     CASE OP_Arr_OP10P[Output_Page_num] OF	
     300: OLine2:= "O10A_SPARE_Q300_1(Q300.1)                   ";
     301: OLine2:= "O10A_BDY_EMPT_CAM_LGHT2_ON(Q301.1)          ";
     302: OLine2:= "O10B_DRUM_RST(Q302.1)                       ";
     303: OLine2:= "O10B_SPARE_Q303_1(Q303.1)                   ";
     304: OLine2:= "O20_SPARE_Q304_1(Q304.1)                    ";
     305: OLine2:= "O30_CAM_LGHT1_ON(Q305.1)                    ";
     306: OLine2:= "O50_SPARE_Q306_1(Q306.1)                    ";
     307: OLine2:= "O70_DRUM_MTR_FWD(Q307.1)                    ";
     308: OLine2:= "O70_BARLIGHT_OP2(Q308.1)                    ";
     309: OLine2:= "O70_SPARE_Q309_1(Q309.1)                    ";
     1050:OLine2:= "O10A_ORING_LH_PUSHR_CYL_REV_FWD(Q1050.1)    ";
     1051:OLine2:= "O10A_ORING_VERT_CYL_DWN(Q1051.1)            ";
     1052:OLine2:= "O10A_DRUM_FEED_AIRPURGE_ON(Q1052.1)         ";
     1053:OLine2:= "O10A_SPARE_Q1053_1(Q1053.1)                 ";
     1060:OLine2:= "O10B_ORING_LH_PUSHR_CYL_REV_FWD(Q1060.1)    ";
     1061:OLine2:= "O10B_ORING_VERT_CYL_DWN(Q1061.1)            ";
     1062:OLine2:= "O10B_SPARE_Q1062_1(Q1062.1)                 ";
     1063:OLine2:= "O10B_SPARE_Q1063_1(Q1063.1)                 ";
     1150:OLine2:= "O20_LH_OIL_SPIN_ON(Q1150.1)                 ";
     1151:OLine2:= "O40_TOOL_CHO_LOCK(Q1151.1)                  ";
     1152:OLine2:= "O50_SPARE_Q1152_1(Q1152.1)                  ";
     1153:OLine2:= "O80_TOOL_CHO_LOCK(Q1153.1)                     ";
     ELSE 
     OLine2 := " ";
     END_CASE
	 Out_Visibility_2:=TRUE;	
    CASE OP_Arr_OP10P[Output_Page_num] OF
	300:  Out_Lamp2:=O10A_SPARE_Q300_1;
	301:  Out_Lamp2:=O10A_BDY_EMPT_CAM_LGHT2_ON_Q301_1;
	302:  Out_Lamp2:=O10B_DRUM_RST_Q302_1;
	303:  Out_Lamp2:=O10B_SPARE_Q303_1;
	304:  Out_Lamp2:=O20_SPARE_Q304_1;
	305:  Out_Lamp2:=O30_CAM_LGHT1_ON_Q305_1;
	306:  Out_Lamp2:=O50_SPARE_Q306_1;
	307:  Out_Lamp2:=O70_DRUM_MTR_FWD_Q307_1;
	308:  Out_Lamp2:=O70_BARLIGHT_OP2_Q308_1;
	309:  Out_Lamp2:=O70_SPARE_Q309_1;
        1050: Out_Lamp2:=O10A_ORING_LH_PUSHR_CYL_REV_FWD_Q1050_1;
	1051: Out_Lamp2:=O10A_ORING_VERT_CYL_DWN_Q1051_1;
	1052: Out_Lamp2:=O50_RH_REJ_CYL_FWD_Q1152_1;
	1053: Out_Lamp2:=O10A_SPARE_Q1053_1;
	1060: Out_Lamp2:=O10B_ORING_LH_PUSHR_CYL_REV_FWD_Q1060_1;
	1061: Out_Lamp2:=O10B_ORING_VERT_CYL_DWN_Q1061_1;
	1062: Out_Lamp2:=O10B_SPARE_Q1062_1;
	1063: Out_Lamp2:=O10B_SPARE_Q1063_1;
	1150: Out_Lamp2:=O20_LH_OIL_SPIN_ON_Q1150_1;
	1151: Out_Lamp2:=O40_TOOL_CHO_LOCK_Q1151_1;
	1152: Out_Lamp2:=O50_RH_REJ_CYL_FWD_Q1152_1;
	1153: Out_Lamp2:=O80_TOOL_CHO_LOCK_Q1153_1;
   ELSE
       Out_Visibility_2:=FALSE;	
   END_CASE 
   
     CASE OP_Arr_OP10P[Output_Page_num] OF	
     300: OLine3:= "O10A_SPARE_Q300_2(Q300.2)		     ";
     301: OLine3:= "O10A_FIRTREE_ORING_CAM_LGHT1_ON(Q301.2)  ";
     302: OLine3:= "O10B_DRUM_EXT_SPEED(Q302.2)              ";
     303: OLine3:= "O10B_FIRTREE_ORING_CAM_LGHT1_ON(Q303.2)  ";
     304: OLine3:= "O20_SPARE_Q304_2(Q304.2)                 ";
     305: OLine3:= "O30_CAM_LGHT2_ON(Q305.2)                 ";
     306: OLine3:= "O50_DRUM_RUN_IND(Q306.2)                 ";
     307: OLine3:= "O70_DRUM_RST(Q307.2)                     ";
     308: OLine3:= "O70_SPARE_Q308_2(Q308.2)                 ";
     309: OLine3:= "O70_SPARE_Q309_2(Q309.2)                 ";
     1050:OLine3:= "O10A_ORING_RH_GRPR_CLSE_OPN(Q1050.2)     ";
     1051:OLine3:= "O10A_LH_FIRTRE_ORING_REJ_CYL_REV(Q1051.2)";
     1052:OLine3:= "O10A_SPARE_Q1052_2(Q1052.2)              ";
     1053:OLine3:= "O10A_SPARE_Q1053_2(Q1053.2)              ";
     1060:OLine3:= "O10B_ORING_RH_GRPR_CLSE_OPN(Q1060.2)     ";
     1061:OLine3:= "O10B_LH_FIRTRE_ORING_REJ_CYL_REV(Q1061.2)";
     1062:OLine3:= "O10B_SPARE_Q1062_2(Q1062.2)              ";
     1063:OLine3:= "O10B_SPARE_Q1063_2(Q1063.2)              ";
     1150:OLine3:= "O20_RH_OIL_DISPN_ON(Q1150_2)             ";
     1151:OLine3:= "O50_LH_GRIP_OPN_CLSE(Q1151.2)            ";
     1152:OLine3:= "O60_TOOL_CHO_UNLOCK(Q1152.2)             ";
     1153:OLine3:= "O30_AIR_PURGE_ON(Q1153.2)                ";
     ELSE
     	OLine3 := " ";
     END_CASE
	 Out_Visibility_3:=TRUE;	
     CASE OP_Arr_OP10P[Output_Page_num] OF
	300:  Out_Lamp3:=O10A_SPARE_Q300_2;
	301:  Out_Lamp3:=O10A_FIRTREE_ORING_CAM_LGHT1_ON_Q301_2;
	302:  Out_Lamp3:=O10B_DRUM_EXT_SPEED_Q302_2;
	303:  Out_Lamp3:=O10B_FIRTREE_ORING_CAM_LGHT1_ON_Q303_2;
	304:  Out_Lamp3:=O20_SPARE_Q304_2;
	305:  Out_Lamp3:=O30_CAM_LGHT2_ON_Q305_2;
	306:  Out_Lamp3:=O50_DRUM_RUN_IND_Q306_2;
	307:  Out_Lamp3:=O70_DRUM_RST_Q307_2;
	308:  Out_Lamp3:=O70_SPARE_Q308_2;
	309:  Out_Lamp3:=O70_SPARE_Q309_2;
    1050: Out_Lamp3:= O10A_ORING_RH_GRPR_CLSE_OPN_Q1050_2;
	1051: Out_Lamp3:=O10A_LH_FIRTRE_ORING_REJ_CYL_REV_Q1051_2;
	1052: Out_Lamp3:=O10A_SPARE_Q1052_2;
	1053: Out_Lamp3:=O10A_SPARE_Q1053_2;
	1060: Out_Lamp3:=O10B_ORING_RH_GRPR_CLSE_OPN_Q1060_2;
	1061: Out_Lamp3:=O10B_LH_FIRTRE_ORING_REJ_CYL_REV_Q1061_2;
	1062: Out_Lamp3:=O10B_SPARE_Q1062_2;
	1063: Out_Lamp3:=O10B_SPARE_Q1063_2;
	1150: Out_Lamp3:=O20_RH_OIL_DISPN_ON_Q1150_2;
	1151: Out_Lamp3:=O50_LH_GRIP_OPN_Q1151_2;
	1152: Out_Lamp3:=O60_TOOL_CHO_UNLOCK_Q1152_2;
	1153: Out_Lamp3:=O30_AIR_PURGE_ON_Q1153_2;
   ELSE
       Out_Visibility_3:=FALSE;	
   END_CASE 
   
     CASE OP_Arr_OP10P[Output_Page_num] OF	
     300: OLine4:= "O10A_SPARE_Q300_3(Q300.3)	           "; 
     301: OLine4:= "O10A_FIRTREE_ORING_CAM_LGHT2_ON(Q301.3)";
     302: OLine4:= "O10A_SPARE_Q302_3(Q302.3)              ";
     303: OLine4:= "O10B_FIRTREE_ORING_CAM_LGHT2_ON(Q303.3)";
     304: OLine4:= "O20_SPARE_Q304_3(Q304.3)               ";
     305: OLine4:= "O30_SPARE_Q305_3(Q305.3)               ";
     306: OLine4:= "O50_CAM_LGHT1_ON(Q306.3)               ";
     307: OLine4:= "O70_DRUM_EXT_SPEED(Q307.3)             ";
     308: OLine4:= "O70_SPARE_Q308_3(Q308.3)               ";
     309: OLine4:= "O70_SPARE_Q309_3(Q309.3)               ";
     1050:OLine4:= "O10A_ORING_RH_PUSHR_CYL_REV_FWD(Q1050.3)";
     1051:OLine4:= "O10A_LH_FIRTRE_ORING_REJ_CYL_FWD(Q1051.3)";
     1052:OLine4:= "O10A_SPARE_Q1052_3(Q1052.3)            ";
     1053:OLine4:= "O10A_SPARE_Q1053_3(Q1053.3)            ";
     1060:OLine4:= "O10B_ORING_RH_PUSHR_CYL_REV_FWD(Q1060.3)";
     1061:OLine4:= "O10B_LH_FIRTRE_ORING_REJ_CYL_FWD(Q1061.3)";
     1062:OLine4:= "O10B_SPARE_Q1062_3(Q1062.3)            ";
     1063:OLine4:= "O10B_SPARE_Q1063_3(Q1063.3)            ";
     1150:OLine4:= "O20_RH_OIL_SPIN_ON(Q1150.3)            ";
     1151:OLine4:= "O50_SPARE_Q1151_3(Q1151.3)             ";
     1152:OLine4:= "O60_TOOL_CHO_LOCK(Q1152.3)             ";
     1153:OLine4:= "O70_SPARE_Q1153_3(Q1153.3)             ";
     ELSE
     	OLine4 := " ";
     END_CASE
       Out_Visibility_4:=TRUE;	
     CASE OP_Arr_OP10P[Output_Page_num] OF
     300:  Out_Lamp4:=O10A_SPARE_Q300_3;
     301:  Out_Lamp4:=O10A_FIRTREE_ORING_CAM_LGHT2_ON_Q301_3;
     302:  Out_Lamp4:=O10A_SPARE_Q302_3_Q302_3;
     303:  Out_Lamp4:=O10B_FIRTREE_ORING_CAM_LGHT2_ON_Q303_3;
     304:  Out_Lamp4:=O20_SPARE_Q304_3;
     305:  Out_Lamp4:=O30_SPARE_Q305_3;
     306:  Out_Lamp4:=O50_CAM_LGHT1_ON_Q306_3;
     307:  Out_Lamp4:=O70_DRUM_EXT_SPEED_Q307_3;
     308:  Out_Lamp4:=O70_SPARE_Q308_3;
     309:  Out_Lamp4:=O70_SPARE_Q309_3;
     1050: Out_Lamp4:=O10A_ORING_RH_PUSHR_CYL_REV_FWD_Q1050_3;
     1051: Out_Lamp4:=O10A_LH_FIRTRE_ORING_REJ_CYL_FWD_Q1051_3;
     1052: Out_Lamp4:=O10A_SPARE_Q1052_3;
     1053: Out_Lamp4:=O10A_SPARE_Q1053_3;
     1060: Out_Lamp4:=O10B_ORING_RH_PUSHR_CYL_REV_FWD_Q1060_3;
     1061: Out_Lamp4:=O10B_LH_FIRTRE_ORING_REJ_CYL_FWD_Q1061_3;
     1062: Out_Lamp4:=O10B_SPARE_Q1062_3;
     1063: Out_Lamp4:=O10B_SPARE_Q1063_3;
     1150: Out_Lamp4:=O20_RH_OIL_SPIN_ON_Q1150_3;
     1151: Out_Lamp4:=O50_LH_GRIP_CLSE_Q1151_3;
     1152: Out_Lamp4:=O60_TOOL_CHO_LOCK_Q1152_3;
     1153: Out_Lamp4:=O30_SPARE_Q1153_3;
     ELSE	
       Out_Visibility_4:=FALSE;	
     END_CASE 
	 
     CASE OP_Arr_OP10P[Output_Page_num] OF	
     300: OLine5:= "O10A_SPARE_Q300_4(Q300.4)	       	     ";
     301: OLine5:= "O10A_ORING_CAM_LGHT1_ON(Q301.4)          ";
     302: OLine5:= "O10B_DRUM_RUN_IND(Q302.4)                ";
     303: OLine5:= "O10B_ORING_CAM_LGHT1_ON(Q303.4)          ";
     304: OLine5:= "O30_DRUM_MTR_FWD(Q304.4)                 ";
     305: OLine5:= "O30_SPARE_Q305_4(Q305.4)                 ";
     306: OLine5:= "O50_CAM_LGHT2_ON(Q306.4)                 ";
     307: OLine5:= "O70_SPARE_Q307_4(Q307.4)                 ";
     308: OLine5:= "O70_SPARE_Q308_4(Q308.4)                 ";
     309: OLine5:= "O70_SPARE_Q309_4(Q309.4)                 ";
     1050:OLine5:= "O10A_ORING_ROTRY_CYL_O_DEG(Q1050.4)      ";
     1051:OLine5:= "O10A_RH_FIRTRE_ORING_REJ_CYL_REV(Q1051.4)";
     1052:OLine5:= "O10A_SPARE_Q1052_4(Q1052.4)              ";
     1053:OLine5:= "O10A_SPARE_Q1053_4(Q1053.4)              ";
     1060:OLine5:= "O10B_ORING_ROTRY_CYL_O_DEG(Q1060.4)      ";
     1061:OLine5:= "O10B_RH_FIRTRE_ORING_REJ_CYL_REV(Q1061.4)";
     1062:OLine5:= "O10B_SPARE_Q1062_4(Q1062.4)              ";
     1063:OLine5:= "O10B_SPARE_Q1063_4(Q1063.4)              ";
     1150:OLine5:= "O30_LH_REJ_CYL_REV(Q1150.4)              ";
     1151:OLine5:= "O50_RH_GRIP_OPN_CLSE(Q1151.4)            ";
     1152:OLine5:= "O70_LH_REJ_CYL_FWD_REV(Q1152.4)          ";
     1153:OLine5:= "O50_AIR_PURGE_ON(Q1153.4)                ";
     ELSE
     	OLine5 := " ";
     END_CASE
         Out_Visibility_5:=TRUE;	
	 CASE OP_Arr_OP10P[Output_Page_num] OF
	      300:  Out_Lamp5:=O10A_SPARE_Q300_4;
	      301:  Out_Lamp5:=O10A_ORING_CAM_LGHT1_ON_Q301_4;
	      302:  Out_Lamp5:=O10B_DRUM_RUN_IND_Q302_4;
	      303:  Out_Lamp5:=O10B_ORING_CAM_LGHT1_ON_Q303_4;
	      304:  Out_Lamp5:=O30_DRUM_MTR_FWD_Q304_4;
	      305:  Out_Lamp5:=O30_SPARE_Q305_4;
	      306:  Out_Lamp5:=O50_CAM_LGHT2_ON_Q306_4;
	      307:  Out_Lamp5:=O70_SPARE_Q307_4;
           308:  Out_Lamp5:=O70_SPARE_Q308_4;
           309:  Out_Lamp5:=O70_SPARE_Q309_4;
	      1050: Out_Lamp5:=O10A_ORING_ROTRY_CYL_O_DEG_Q1050_4;
	      1051: Out_Lamp5:=O10A_RH_FIRTRE_ORING_REJ_CYL_REV_Q1051_4;
	      1052: Out_Lamp5:=O10A_SPARE_Q1052_4;
	      1053: Out_Lamp5:=O10A_SPARE_Q1053_4;
	      1060: Out_Lamp5:=O10B_ORING_ROTRY_CYL_O_DEG_Q1060_4;
	      1061: Out_Lamp5:=O10B_RH_FIRTRE_ORING_REJ_CYL_REV_Q1061_4;
	      1062: Out_Lamp5:=O10B_SPARE_Q1062_4;
	      1063: Out_Lamp5:=O10B_SPARE_Q1063_4;
	      1150: Out_Lamp5:=O30_LH_REJ_CYL_REV_Q1150_4;
	      1151: Out_Lamp5:=O50_RH_GRIP_OPN_Q1151_4;
	      1152: Out_Lamp5:=O70_LH_REJ_CYL_REV_Q1152_4;
	      1153: Out_Lamp5:=O50_AIR_PURGE_ON_Q1153_4;
 	      ELSE
    	        Out_Visibility_5:=FALSE;	
  	      END_CASE
	 
     CASE OP_Arr_OP10P[Output_Page_num] OF	
     300: OLine6:= "O10A_SPARE_Q300_5(Q300.5)					";
     301: OLine6:= "O10A_ORING_CAM_LGHT2_ON(Q301.5)          ";
     302: OLine6:= "O10_TWR_LMP_RD(Q302.5)                  ";
     303: OLine6:= "O10B_ORING_CAM_LGHT2_ON(Q303.5)          ";
     304: OLine6:= "O30_DRUM_RST(Q304.5)                      ";
     305: OLine6:= "O50_DRUM_MTR_FWD(Q305.5)                  ";
     306: OLine6:= "O50_SPARE_Q306_5(Q306.5)                  ";
     307: OLine6:= "O70_DRUM_RUN_IND(Q307.5)                  ";
     308: OLine6:= "O70_SPARE_Q308_5(Q308.5)                  ";
     309: OLine6:= "O70_SPARE_Q309_5(Q309.5)                  ";
     1050:OLine6:= "O10A_ORING_ROTRY_CYL_180_DEG(Q1050.5)     ";
     1051:OLine6:= "O10A_RH_FIRTRE_ORING_REJ_CYL_FWD(Q1051.5) ";
     1052:OLine6:= "O10A_SPARE_Q1052_5(Q1052.5)               ";
     1053:OLine6:= "O10A_SPARE_Q1053_5(Q1053.5)               ";
     1060:OLine6:= "O10B_ORING_ROTRY_CYL_180_DEG(Q1060.5)     ";
     1061:OLine6:= "O10B_RH_FIRTRE_ORING_REJ_CYL_FWD(Q1061.5) ";
     1062:OLine6:= "O10B_SPARE_Q1062_5	(Q1062.5)             ";
     1063:OLine6:= "O10B_SPARE_Q1063_5	(Q1063.5)             ";
     1150:OLine6:= "O30_LH_REJ_CYL_FWD	(Q1150.5)             ";
     1151:OLine6:= "O50_SPARE_Q1151_5	(Q1151.5)             ";
     1152:OLine6:= "O70_SPARE_Q1152_5	(Q1152.5)             ";
     1153:OLine6:= "O70_AIR_PURGE_ON	Q1153.5               ";
     ELSE
     	OLine6 := " ";
     END_CASE
	 
     Out_Visibility_6:=TRUE;	
	 CASE OP_Arr_OP10P[Output_Page_num] OF
	300:  Out_Lamp6:=O10A_SPARE_Q300_5;
	301:  Out_Lamp6:=O10A_ORING_CAM_LGHT2_ON_Q301_5;
	302:  Out_Lamp6:=O10_TWR_LMP_RD_Q302_5;
	303:  Out_Lamp6:=O10B_ORING_CAM_LGHT2_ON_Q303_5;
	304:  Out_Lamp6:=O30_DRUM_RST_Q304_5;
	305:  Out_Lamp6:=O50_DRUM_MTR_FWD_Q305_5;
	306:  Out_Lamp6:=O50_SPARE_Q306_5;
	307:  Out_Lamp6:=O70_DRUM_RUN_IND_Q307_5;
	308:  Out_Lamp6:=O70_SPARE_Q308_5;
	309:  Out_Lamp6:=O70_SPARE_Q309_5;
	1050: Out_Lamp6:=O10A_ORING_ROTRY_CYL_180_DEG_Q1050_5;
	1051: Out_Lamp6:=O10A_RH_FIRTRE_ORING_REJ_CYL_FWD_Q1051_5;
	1052: Out_Lamp6:=O10A_SPARE_Q1052_5;
	1053: Out_Lamp6:=O10A_SPARE_Q1053_5;
	1060: Out_Lamp6:=O10B_ORING_ROTRY_CYL_180_DEG_Q1060_5;
	1061: Out_Lamp6:=O10B_RH_FIRTRE_ORING_REJ_CYL_FWD_Q1061_5;
	1062: Out_Lamp6:=O10B_SPARE_Q1062_5;
	1063: Out_Lamp6:=O10B_SPARE_Q1063_5;
	1150: Out_Lamp6:=O30_LH_REJ_CYL_FWD_Q1150_5;
	1151: Out_Lamp6:=O50_RH_GRIP_CLSE_Q1151_5;
	1152: Out_Lamp6:=O70_LH_REJ_CYL_FWD_Q1152_5;
	1153: Out_Lamp6:=O30_SPARE_Q1153_5;
   ELSE           
       Out_Visibility_6:=FALSE;	
   END_CASE
	 
     CASE OP_Arr_OP10P[Output_Page_num] OF	
     300: OLine7:= "O10_BARLIGHT_OP1(Q300.6)                      ";
     301: OLine7:= "O10A_FIRTREE_ORING_CAMBAR_LGHT1_ON(Q301.6)    ";
     302: OLine7:= "O10_TWR_LMP_GN(Q302.6)                        ";
     303: OLine7:= "O10B_FIRTREE_ORING_CAMBAR_LGHT1_ON(Q303.6)    ";
     304: OLine7:= "O30_DRUM_EXT_SPEED(Q304.6)                    ";
     305: OLine7:= "O50_DRUM_RST(Q305.6)                          ";
     306: OLine7:= "O50_SPARE_Q306_6(Q306.6)                      ";
     307: OLine7:= "O70_CAM_LGHT1_ON(Q307.6)                      ";
     308: OLine7:= "O70_SPARE_Q308_6(Q308.6)                      ";
     309: OLine7:= "O70_SPARE_Q309_6(Q309.6)                      ";
     1050:OLine7:= "O10A_ORING_HORZ_CYL_REV(Q1050.6)              ";
     1051:OLine7:= "O10A_BDY_SING_CYL_CLSE(Q1051.6)               ";
     1052:OLine7:= "O10A_SPARE_Q1052_6(Q1052.6)                   ";
     1053:OLine7:= "O10A_SPARE_Q1053_6(Q1053.6)                   ";
     1060:OLine7:= "O10B_ORING_HORZ_CYL_REV(Q1060.6)              ";
     1061:OLine7:= "O10B_BDY_SING_CYL_CLSE(Q1061.6)               ";
     1062:OLine7:= "O10B_SPARE_Q1062_6(Q1062.6)                   ";
     1063:OLine7:= "O10B_SPARE_Q1063_6(Q1063.6)                   ";
     1150:OLine7:= "O30_RH_REJ_CYL_REV(Q1150.6)                   ";
     1151:OLine7:= "O50_LH_REJ_CYL_FWD_REV(Q1151.6)               ";
     1152:OLine7:= "O70_RH_REJ_CYL_FWD_REV(Q1152.6)               ";
     1153:OLine7:= "O80_SPARE_Q1153_6(Q1153.6)                    ";
     ELSE
     	OLine7 := " ";
     END_CASE
     
	 Out_Visibility_7:=TRUE;	
	 CASE OP_Arr_OP10P[Output_Page_num] OF
	300:  Out_Lamp7:=O10_BARLIGHT_OP1_Q300_6;
	301:  Out_Lamp7:=O10A_FIRTREE_ORING_CAMBAR_LGHT1_ON_Q301_6;
	302:  Out_Lamp7:=O10_TWR_LMP_GN_Q302_6;
	303:  Out_Lamp7:=O10B_FIRTREE_ORING_CAMBAR_LGHT1_ON_Q303_6;
	304:  Out_Lamp7:=O30_DRUM_EXT_SPEED_Q304_6;
	305:  Out_Lamp7:=O50_DRUM_RST_Q305_6;
	306:  Out_Lamp7:=O50_SPARE_Q306_6;
	307:  Out_Lamp7:=O70_CAM_LGHT1_ON_Q307_6;
	308:  Out_Lamp7:=O70_SPARE_Q308_6;
	309:  Out_Lamp7:=O70_SPARE_Q309_6;
	1050: Out_Lamp7:=O10A_ORING_HORZ_CYL_REV_Q1050_6;
	1051: Out_Lamp7:=O10A_BDY_SING_CYL_CLSE_Q1051_6;
	1052: Out_Lamp7:=O10A_SPARE_Q1052_6;
	1053: Out_Lamp7:=O10A_SPARE_Q1053_6;
	1060: Out_Lamp7:=O10B_ORING_HORZ_CYL_REV_Q1060_6;
	1061: Out_Lamp7:=O10B_BDY_SING_CYL_CLSE_Q1061_6;
	1062: Out_Lamp7:=O10B_SPARE_Q1062_6;
	1063: Out_Lamp7:=O10B_SPARE_Q1063_6;
	1150: Out_Lamp7:=O30_RH_REJ_CYL_REV_Q1150_6;
	1151: Out_Lamp7:=O50_LH_REJ_CYL_REV_Q1151_6;
	1152: Out_Lamp7:=O70_RH_REJ_CYL_REV_Q1152_6;
	1153: Out_Lamp7:=O70_AIR_PURGE_ON_Q1153_6;
   ELSE
       Out_Visibility_7:=FALSE;	
   END_CASE 
	 
     CASE OP_Arr_OP10P[Output_Page_num] OF	
     300: OLine8:= "O10_BARLIGHT_OP2(Q300.7)	       ";
     301: OLine8:= "O10A_SPARE_Q301_7(Q301.7)          ";
     302: OLine8:= "O10_TWR_LMP_YELW(Q302.7)           ";
     303: OLine8:= "O10B_SPARE_Q303_7(Q303.7)          ";
     304: OLine8:= "O30_SPARE_Q304_7(Q304.7)           ";
     305: OLine8:= "O50_SPARE_Q305_7(Q305.7)           ";
     306: OLine8:= "O50_BARLIGHT_OP1(Q306.7)           ";
     307: OLine8:= "O70_CAM_LGHT2_ON(Q307.7)           ";
     308: OLine8:= "O70_SPARE_Q308_7(Q308.7)           ";
     309: OLine8:= "O70_SPARE_Q309_7(Q309.7)           ";
     1050:OLine8:= "O10A_ORING_HORZ_CYL_FWD(Q1050.7)   ";
     1051:OLine8:= "O10A_BDY_SING_CYL_OPN(Q1051.7)     ";
     1052:OLine8:= "O10A_SPARE_Q1052_7(Q1052.7)        ";
     1053:OLine8:= "O10A_SPARE_Q1053_7(Q1053.7)        ";
     1060:OLine8:= "O10B_ORING_HORZ_CYL_FWD(Q1060.7)   ";
     1061:OLine8:= "O10B_BDY_SING_CYL_OPN(Q1061.7)     ";
     1062:OLine8:= "O10B_SPARE_Q1062_7(Q1062.7)        ";
     1063:OLine8:= "O10B_SPARE_Q1063_7(Q1063.7)        ";
     1150:OLine8:= "O30_RH_REJ_CYL_FWD(Q1150.7)        ";
     1151:OLine8:= "O50_SPARE_Q1151_7(Q1151.7)         ";
     1152:OLine8:= "O70_SPARE_Q1152_7(Q1152.7)         ";
     1153:OLine8:= "O80_SPARE_Q1153_7(Q1153.7)         ";
     ELSE
     	OLine8 := " ";
     END_CASE
	 Out_Visibility_8:=TRUE;	
	 CASE OP_Arr_OP10P[Output_Page_num] OF
	300:  Out_Lamp8:=O10_BARLIGHT_OP2_Q300_7;
	301:  Out_Lamp8:=O10A_SPARE_Q301_7;
	302:  Out_Lamp8:=O10_TWR_LMP_YELW_Q302_7;
	303:  Out_Lamp8:=O10B_SPARE_Q303_7;
	304:  Out_Lamp8:=O30_SPARE_Q304_7_Q304_7;
	305:  Out_Lamp8:=O50_SPARE_Q305_7;
	306:  Out_Lamp8:=O50_BARLIGHT_OP1_Q306_7;
	307:  Out_Lamp8:=O70_CAM_LGHT2_ON_Q307_7;
	308:  Out_Lamp8:=O70_SPARE_Q308_7;
	309:  Out_Lamp8:=O70_SPARE_Q309_7;
	1050: Out_Lamp8:=O10A_ORING_HORZ_CYL_FWD_Q1050_7;
	1051: Out_Lamp8:=O10A_BDY_SING_CYL_OPN_Q1051_7;
	1052: Out_Lamp8:=O10A_SPARE_Q1052_7;
	1053: Out_Lamp8:=O10A_SPARE_Q1053_7;
	1060: Out_Lamp8:=O10B_ORING_HORZ_CYL_FWD_Q1060_7;
	1061: Out_Lamp8:=O10B_BDY_SING_CYL_OPN_Q1061_7;
	1062: Out_Lamp8:=O10B_SPARE_Q1062_7;
	1063: Out_Lamp8:=O10B_SPARE_Q1063_7;
	1150: Out_Lamp8:=O30_RH_REJ_CYL_FWD_Q1150_7;
	1151: Out_Lamp8:=O50_LH_REJ_CYL_FWD_Q1151_7;
	1152: Out_Lamp8:=O70_RH_REJ_CYL_FWD_Q1152_7;
	1153: Out_Lamp8:=O30_SPARE_Q1153_7;
   ELSE
       Out_Visibility_8:=FALSE;	
   END_CASE  
	 
 2: CASE IP_Arr_OP90P[Input_Page_num] OF
   400:  Line1:= " I90_PMR_FB(I400.0)                   ";
   401:  Line1:= " I90_DOOR7_CLOSE_FB(I401.0)           ";
   402:  Line1:= " I90_DOOR15_CLOSE_FB(I402.0)          ";
   403:  Line1:= " I120_ATC_STN_POKE_YOKE_3(I403.0)     ";
   404:  Line1:="I90_LHS_ESTOP1_FB(I404.0)	      "  ;
   405:  Line1:="I90_XTS_48VSMPS1_DC_OK(I405.0)        " ;
   1200: Line1:= " I90_RET_LH_GRIPR_CYL_CLSE(I1200.0)   ";
   1201: Line1:= " I90_LH_MOVR_SUP_HORZ_CYL_REV(I1201.0)";
   1210: Line1:= " I90_LH1_REJ_SLIDE_REV(I1210.0)       ";
   1211: Line1:= " I90_SPARE_I1211_0(I1211.0)           ";
   1220: Line1:= " I120_PUSH_CYL_REV(I1220.0)           ";
   1221: Line1:= " I120_REJ_BIN_PRSNCE(I1221.0)          ";
   ELSE
     Line1:= " ";	
   END_CASE
   Visibility_1:=TRUE;
   
   CASE IP_Arr_OP90P[Input_Page_num] OF
	400: Lamp1:=I90_PMR_FB_I400_0 ;
	401: Lamp1:=I90_DOOR7_CLOSE_FB_I401_0 ;
	402: Lamp1:=I90_DOOR15_CLOSE_FB_I402_0 ;
	403: Lamp1:=I120_ATC_STN_POKE_YOKE_3_I403_0;
	404: Lamp1:=I90_LHS_ESTOP1_FB_I404_0 ;
	405: Lamp1:=I90_XTS_48VSMPS1_DC_OK_I405_0 ;
	1200: Lamp1:=I90_RET_LH_GRIPR_CYL_CLSE_I1200_0 ;
	1201: Lamp1:=I90_LH_MOVR_SUP_HORZ_CYL_REV_I1201_0 ;
	1210: Lamp1:=I90_LH1_REJ_SLIDE_REV_I1210_0;
	1211: Lamp1:=I90_SPARE_I1211_0;
	1220: Lamp1:=I120_PUSH_CYL_REV_I1220_0 ;
	1221: Lamp1:=I120_REJ_BIN_PRSNCE_I1221_0 ;
   ELSE
       Visibility_1:=FALSE;	
   END_CASE
   
   CASE IP_Arr_OP90P[Input_Page_num] OF
   400:  Line2:= " I90_SURGE_ARRES_FB(I400.1)           ";
   401:  Line2:= " I90_DOOR8_CLOSE_FB(I401.1)           ";
   402:  Line2:= " I90_DOOR16_CLOSE_FB(I402.1)          ";
   403:  Line2:= " I120_ATC_STN_POKE_YOKE_4(I403.1)     ";
   404: Line2:="I90_LHS_ESTOP2_FB(I404.1)             " ;
   405: Line2:="I90_XTS_48VSMPS2_DC_OK(I405.1)        " ;
   1200: Line2:= " I90_RET_LH_GRIPR_CYL_OPN(I1200.1)    ";
   1201: Line2:= " I90_LH_MOVR_SUP_HORZ_CYL_FWD(I1201.1)";
   1210: Line2:= " I90_LH1_REJ_SLIDE_FWD(I1210.1)       ";
   1211: Line2:= " I90_SPARE_I1211_1(I1211.1)           ";
   1220: Line2:= " I120_PUSH_CYL_FWD(I1220.1)           ";
   1221: Line2:= " I120_SPARE_I1221_1(I1221.1)          ";
   ELSE
     Line2:= " ";	
   END_CASE
     
   Visibility_2:=TRUE;
   
   CASE IP_Arr_OP90P[Input_Page_num] OF
	400: Lamp2:=I90_SURGE_ARRES_FB_I400_1  ;
	401: Lamp2:=I90_DOOR8_CLOSE_FB_I401_1 ;
	402: Lamp2:=I90_DOOR16_CLOSE_FB_I402_1 ;
	403: Lamp2:=I120_ATC_STN_POKE_YOKE_4_I403_1;
	404: Lamp2:=I90_LHS_ESTOP2_FB_I404_1 ;
	405: Lamp2:=I90_XTS_48VSMPS2_DC_OK_I405_1 ;
	1200:Lamp2:=I90_RET_LH_GRIPR_CYL_OPN_I1200_1;
	1201:Lamp2:=I90_LH_MOVR_SUP_HORZ_CYL_FWD_I1201_1  ;
	1210:Lamp2:=I90_LH1_REJ_SLIDE_FWD_I1210_1;
	1211:Lamp2:=I90_SPARE_I1211_1 ;
	1220:Lamp2:=I120_PUSH_CYL_FWD_I1220_1 ;
	1221:Lamp2:=I120_SPARE_I1221_1 ;
   ELSE
       Visibility_2:=FALSE;	
   END_CASE
   
   CASE IP_Arr_OP90P[Input_Page_num] OF
   400:  Line3:= " I90_DOOR1_CLOSE_FB(I400.2)           ";
   401:  Line3:= " I90_DOOR9_CLOSE_FB(I401.2)           ";
   402:  Line3:= " I110_RESRVR_LW_LVL(I402.2)           ";
   403:  Line3:= " I120_ATC_SLAVE_MODL1(I403.2)         ";
   404:  Line3:= "I90_LHS_ESTOP3_FB(I404.2)             " ;
   405:  Line3:= "I90_XTS_48VSMPS3_DC_OK(I405.2)        " ;
   1200: Line3:= " I90_RET_RH_GRIPR_CYL_CLSE(I1200.2)   ";
   1201: Line3:= " I90_RH_MOVR_SUP_VERT_CYL_DWN(I1201.2)";
   1210: Line3:= " I90_RH1_REJ_SLIDE_REV(I1210.2)       ";
   1211: Line3:= " I90_SPARE_I1211_2(I1211.2)           ";
   1220: Line3:= " I120_LH_SING_CYL_REV(I1220.2)        ";
   1221: Line3:= " I120_SPARE_I1221_2(I1221.2)          ";
   ELSE
     Line3:= " ";	
   END_CASE
  
    Visibility_3:=TRUE;
   
   CASE IP_Arr_OP90P[Input_Page_num] OF
	400: Lamp3:=I90_DOOR1_CLOSE_FB_I400_2  ;
	401: Lamp3:=I90_DOOR9_CLOSE_FB_I401_2 ;
	402: Lamp3:=I110_RESRVR_LW_LVL_I402_2 ;
	403: Lamp3:=I120_ATC_SLAVE_MODL1_I403_2 ;
	404: Lamp3:=I90_LHS_ESTOP3_FB_I404_2 ;
	405: Lamp3:=I90_XTS_48VSMPS3_DC_OK_I405_2;
	1200:Lamp3:=I90_RET_RH_GRIPR_CYL_CLSE_I1200_2;
	1201:Lamp3:=I90_RH_MOVR_SUP_VERT_CYL_DWN_I1201_2 ;
	1210:Lamp3:=I90_RH1_REJ_SLIDE_REV_I1210_2 ;
	1211:Lamp3:=I90_SPARE_I1211_2;
	1220:Lamp3:=I120_LH_SING_CYL_REV_I1220_2 ;
	1221:Lamp3:=I120_SPARE_I1221_2 ;
   ELSE
       Visibility_3:=FALSE;	
   END_CASE
     
   CASE IP_Arr_OP90P[Input_Page_num] OF
   400:  Line4:= " I90_DOOR2_CLOSE_FB(I400.3)          ";
   401:  Line4:= " I90_DOOR10_CLOSE_FB(I401.3)         ";
   402:  Line4:= " I110_OILTANK_PRES_SW_FB(I402.3)     ";
   403:  Line4:= " I120_ATC_SLAVE_MODL2(I403.3)        ";
   404:Line4:="I90_RHS_ESTOP1_FB(I404.3)             " ;
   405:Line4:="I90_XTS_24VSMPS_DC_OK(I405.3)         " ;
   1200: Line4:= " I90_RET_RH_GRIPR_CYL_OPN(I1200.3)   ";
   1201: Line4:= " I90_RH_MOVR_SUP_VERT_CYL_UP(I1201.3)";
   1210: Line4:= " I90_RH1_REJ_SLIDE_FWD(I1210.3)      ";
   1211: Line4:= " I90_SPARE_I1211_3(I1211.3)          ";
   1220: Line4:= " I120_LH_SING_CYL_FWD(I1220.3)       ";
   1221: Line4:= " I120_SPARE_I1221_3(I1221.3)         ";
   ELSE
     Line4:= " ";	
   END_CASE
   Visibility_4:=TRUE;
   
   CASE IP_Arr_OP90P[Input_Page_num] OF
	400: Lamp4:=I90_DOOR2_CLOSE_FB_I400_3   ;
	401: Lamp4:=I90_DOOR10_CLOSE_FB_I401_3;
	402: Lamp4:=I110_OILTANK_PRES_SW_FB_I402_3 ;
	403: Lamp4:=I120_ATC_SLAVE_MODL2_I403_3 ;
	404: Lamp4:=I90_RHS_ESTOP1_FB_I404_3 ;
	405: Lamp4:=I90_XTS_24VSMPS_DC_OK_I405_3;
	1200:Lamp4:=I90_RET_RH_GRIPR_CYL_OPN_I1200_3;
	1201:Lamp4:=I90_RH_MOVR_SUP_VERT_CYL_UP_I1201_3  ;
	1210:Lamp4:=I90_RH1_REJ_SLIDE_FWD_I1210_3;
	1211:Lamp4:=I90_SPARE_I1211_3 ;
	1220:Lamp4:=I120_LH_SING_CYL_FWD_I1220_3;
	1221:Lamp4:=I120_SPARE_I1221_3  ;
   ELSE
       Visibility_4:=FALSE;	
   END_CASE  
   
   
   CASE IP_Arr_OP90P[Input_Page_num] OF
   400:  Line5:= " I90_DOOR3_CLOSE_FB(I400.4)           ";
   401:  Line5:= " I90_DOOR11_CLOSE_FB(I401.4)          ";
   402:  Line5:= " I120_ATC_DECLAMP_FB(I402.4)          ";
   403:  Line5:= " I120_SPARE_I403_4(I403.4)            ";
   404:Line5:="I90_RHS_ESTOP2_FB(I404.4)             " ;
   405:Line5:="I120_LH_LOCKSPRING_GRPR_CLSE(I405.4)  " ;
   1200: Line5:= " I90_POSTN_SLIDE_CYL_REV(I1200.4)     ";
   1201: Line5:= " I90_RH_MOVR_SUP_HORZ_CYL_REV(I1201.4)";
   1210: Line5:= " I90_LH2_REJ_SLIDE_REV(I1210.4)       ";
   1211: Line5:= " I90_SPARE_I1211_4(I1211.4)           ";
   1220: Line5:= " I120_CAMERA_SLIDE_CYL_REV(I1220.4)";
   1221: Line5:= " I120_SPARE_I1221_4(I1221.4)          ";
   ELSE
     Line5:= " ";	
   END_CASE
      
    Visibility_5:=TRUE;
   
   CASE IP_Arr_OP90P[Input_Page_num] OF
	400: Lamp5:=I90_DOOR3_CLOSE_FB_I400_4   ;
	401: Lamp5:=I90_DOOR11_CLOSE_FB_I401_4;
	402: Lamp5:=I120_ATC_DECLAMP_FB_I402_4 ;
	403: Lamp5:=I120_SPARE_I403_4 ;
	404: Lamp5:=I90_RHS_ESTOP2_FB_I404_4 ;
	405: Lamp5:=I120_LH_LOCKSPRING_GRPR_CLSE_I405_4;
	1200:Lamp5:=I90_POSTN_SLIDE_CYL_REV_I1200_4;
	1201:Lamp5:=I90_RH_MOVR_SUP_HORZ_CYL_REV_I1201_4  ;
	1210:Lamp5:=I90_LH2_REJ_SLIDE_REV_I1210_4;
	1211:Lamp5:=I90_SPARE_I1211_4 ;
	1220:Lamp5:=I120_CAMERA_SLIDE_CYL_REV_I1220_4;
	1221:Lamp5:=I120_SPARE_I1221_4 ;
   ELSE
       Visibility_5:=FALSE;	
   END_CASE  
   
   CASE IP_Arr_OP90P[Input_Page_num] OF
   400:  Line6:= " I90_DOOR4_CLOSE_FB(I400.5)            ";
   401:  Line6:= " I90_DOOR12_CLOSE_FB(I401.5)           ";
   402:  Line6:= " I120_ATC_CLAMP_FB(I402.5)             ";
   403:  Line6:= " I120_SPARE_I403_5(I403.5)              ";
   404:Line6:="I90_RHS_ESTOP3_FB(I404.5)             " ;
   405:Line6:="I120_LH_LOCKSPRING_GRPR_OPN(I405.5)   " ;
   1200: Line6:= " I90_POSTN_SLIDE_CYL_FWD(I1200.5)      ";
   1201: Line6:= " I90_RH_MOVR_SUP_HORZ_CYL_FWD(I1201.5) ";
   1210: Line6:= " I90_LH2_REJ_SLIDE_FWD(I1210.5)        ";
   1211: Line6:= " I90_SPARE_I1211_5(I1211.5)            ";
   1220: Line6:= " I120_CAMERA_SLIDECYL_FWD(I1220.5)  ";
   1221: Line6:= " I120_SPARE_I1221_5(I1221.5)           ";
   ELSE
     Line6:= " ";	
   END_CASE
   
     
  Visibility_6:=TRUE;
   
   CASE IP_Arr_OP90P[Input_Page_num] OF
	400: Lamp6:=I90_DOOR4_CLOSE_FB_I400_5 ;
	401: Lamp6:=I90_DOOR12_CLOSE_FB_I401_5;
	402: Lamp6:=I120_ATC_CLAMP_FB_I402_5 ;
	403: Lamp6:=I120_SPARE_I403_5 ;
	404: Lamp6:=I90_RHS_ESTOP3_FB_I404_5 ;
	405: Lamp6:=I120_LH_LOCKSPRING_GRPR_OPN_I405_5;
	1200:Lamp6:=I90_POSTN_SLIDE_CYL_FWD_I1200_5;
	1201:Lamp6:=I90_RH_MOVR_SUP_HORZ_CYL_FWD_I1201_5  ;
	1210:Lamp6:=I90_LH2_REJ_SLIDE_FWD_I1210_5;
	1211:Lamp6:=I90_SPARE_I1211_5 ;
	1220:Lamp6:=I120_CAMERA_SLIDE_CYL_FWD_I1220_5;
	1221:Lamp6:=I120_SPARE_I1221_5  ;
   ELSE
       Visibility_6:=FALSE;	
   END_CASE  
   CASE IP_Arr_OP90P[Input_Page_num] OF
   400:  Line7:= " I90_DOOR5_CLOSE_FB(I400.6)           ";
   401:  Line7:= " I90_DOOR13_CLOSE_FB(I401.6)          ";
   402:  Line7:= " I120_ATC_STN_POKE_YOKE_1(I402.6)     ";
   403:  Line7:= " I120_SPARE_I403_6(I403.6)            ";
   404:Line7:="I90_SPARE_I404_6(I404.6)              " ;
   405:Line7:="I120_RH_LOCKSPRING_GRPR_CLSE(I405.6)  " ;
   1200: Line7:= " I90_LH_MOVR_SUP_VERT_CYL_DWN(I1200.6)";
   1201: Line7:= " I90_SPARE_I1201_6(I1201.6)           ";
   1210: Line7:= " I90_RH2_REJ_SLIDE_REV(I1210.6)       ";
   1211: Line7:= " I90_SPARE_I1211_6(I1211.6)           ";
   1220: Line7:= " I120_SLAVE1_PRSN_PARK_TRAY(I1220.6)";
   1221: Line7:= " I120_SPARE_I1221_6(I1221.6)          ";
   ELSE
     Line7:= " ";	
   END_CASE
   
    Visibility_7:=TRUE;
   
   CASE IP_Arr_OP90P[Input_Page_num] OF
	400: Lamp7:=I90_DOOR5_CLOSE_FB_I400_6 ;
	401: Lamp7:=I90_DOOR13_CLOSE_FB_I401_6;
	402: Lamp7:=I120_ATC_STN_POKE_YOKE_1_I402_6 ;
	403: Lamp7:=I120_SPARE_I403_6 ;
	404: Lamp7:=I90_SPARE_I404_6 ;
	405: Lamp7:=I120_RH_LOCKSPRING_GRPR_CLSE_I405_6;
	1200:Lamp7:=I90_LH_MOVR_SUP_VERT_CYL_DWN_I1200_6;
	1201:Lamp7:=I90_SPARE_I1201_6  ;
	1210:Lamp7:=I90_RH2_REJ_SLIDE_REV_I1210_6;
	1211:Lamp7:=I90_SPARE_I1211_6 ;
	1220:Lamp7:=I120_SLAVE1_PRSN_PARK_TRAY_I1220_6;
	1221:Lamp7:=I120_SPARE_I1221_6  ;
   ELSE
       Visibility_7:=FALSE;	
   END_CASE  
     
   CASE IP_Arr_OP90P[Input_Page_num] OF
   400:  Line8:= " I90_DOOR6_CLOSE_FB(I400.7)          ";
   401:  Line8:= " I90_DOOR14_CLOSE_FB(I401.7)         ";
   402:  Line8:= " I120_ATC_STN_POKE_YOKE_2(I402.7)    ";
   403:  Line8:= " I90_RESET_FB_I403_7I403.7)            ";
   404:Line8:="I90_SPARE_I404_7(I404.7)              " ;
   405:Line8:="I120_RH_LOCKSPRING_GRPR_OPN(I405.7)   " ;
   1200: Line8:= " I90_LH_MOVR_SUP_VERT_CYL_UP(I1200.7)";
   1201: Line8:= " I90_SPARE_I1201_7(I1201.7)          ";
   1210: Line8:= " I90_RH2_REJ_SLIDE_FWD(I1210.7)      ";
   1211: Line8:= " I90_SPARE_I1211_7(I1211.7)          ";
   1220: Line8:= " I120_SLAVE2_PRSN_PARK_TRAY(I1220.7)";
   1221: Line8:= " I120_SPARE_I1221_7(I1221.7)         ";
   ELSE
     Line8:= " ";	
   END_CASE
   
     Visibility_8:=TRUE;
   
   CASE IP_Arr_OP90P[Input_Page_num] OF
	400: Lamp8:=I90_DOOR6_CLOSE_FB_I400_7 ;
	401: Lamp8:=I90_DOOR14_CLOSE_FB_I401_7;
	402: Lamp8:=I120_ATC_STN_POKE_YOKE_2_I402_7 ;
	403: Lamp8:=I90_RESET_FB_I403_7 ;
	404: Lamp8:=I90_SPARE_I404_7 ;
	405: Lamp8:=I120_RH_LOCKSPRING_GRPR_OPN_I405_7;
	1200:Lamp8:=I90_LH_MOVR_SUP_VERT_CYL_UP_I1200_7;
	1201:Lamp8:=I90_SPARE_I1201_7 ;
	1210:Lamp8:=I90_RH2_REJ_SLIDE_FWD_I1210_7;
	1211:Lamp8:=I90_SPARE_I1211_7 ;
	1220:Lamp8:=I120_SLAVE2_PRSN_PARK_TRAY_I1220_7;
	1221:Lamp8:=I120_SPARE_I1221_7   ;
   ELSE
       Visibility_8:=FALSE;	
   END_CASE  
   
    CASE OP_Arr_OP90P[Output_Page_num] OF
    400:  OLine1:= "O90_VISN_LGHT1_ON(Q400.0)            ";
    401:  OLine1:= "O90_SPARE_Q401_0(Q401.0)             ";
    402:  OLine1:= "O110_SPARE_Q402_0(Q402.0)            ";
    403:  OLine1:= "O120_TWR_LMP_RD(Q403.0)              ";
    1240: OLine1:= "O90_RET_LH_GRIPR_CYL_CLSE(Q1240.0)   ";
    1241: OLine1:= "O90_POSTN_SLIDE_CYL_REV(Q1241.0)     ";
    1242: OLine1:= "O90_RH_MOVR_SUP_HORZ_CYL_REV(Q1242.0)";
    1250: OLine1:= "O90_LH1_REJ_SLIDE_REV(Q1250.0)       ";
    1251: OLine1:= "O90_RH2_REJ_SLIDE_REV(Q1251.0)       ";
    1260: OLine1:= "O110_LH_OIL_DISPN_ON(Q1260.0)        ";
    1261: OLine1:= "O120_TOOL_CHO_UNLOCK(Q1261.0)        ";
    1262: OLine1:= "O120_CAMERA_SLIDE_CYL_REV(Q1262.0)   ";
    ELSE
      OLine1:= " ";	
    END_CASE
    Out_Visibility_1:=TRUE;
    CASE OP_Arr_OP90P[Output_Page_num] OF
	400:  Out_Lamp1:=O90_VISN_LGHT1_ON_Q400_0;
	401:  Out_Lamp1:=O90_SPARE_Q401_0;
	402:  Out_Lamp1:=O110_SPARE_Q402_0;
	403:  Out_Lamp1:=O120_TWR_LMP_RD_Q403_0;
    1240:  Out_Lamp1:=O90_RET_LH_GRIPR_CYL_CLSE_Q1240_0;
    1241:  Out_Lamp1:=O90_POSTN_SLIDE_CYL_REV_Q1241_0;
    1242:  Out_Lamp1:=O90_RH_MOVR_SUP_HORZ_CYL_REV_Q1242_0;
    1250:  Out_Lamp1:=O90_LH1_REJ_SLIDE_REV_Q1250_0;
    1251:  Out_Lamp1:=O90_RH2_REJ_SLIDE_REV_Q1251_0;
    1260:  Out_Lamp1:=O110_LH_OIL_DISPN_ON_Q1260_0;
    1261:  Out_Lamp1:=O120_TOOL_CHO_UNLOCK_Q1261_0;
    1262:  Out_Lamp1:=O120_CAMERA_SLIDECYL_REV_Q1262_0;
   ELSE
       Out_Visibility_1:=FALSE;	
   END_CASE
	
    CASE OP_Arr_OP90P[Output_Page_num] OF
    400:  OLine2:= "O90_VISN_LGHT2_ON(Q400.1)            ";
    401:  OLine2:= "O90_SPARE_Q401_1(Q401.1)             ";
    402:  OLine2:= "O110_SPARE_Q402_1(Q402.1)            ";
    403:  OLine2:= "O120_TWR_LMP_GN(Q403.1)              ";
    1240: OLine2:= "O90_RET_LH_GRIPR_CYL_OPN(Q1240.1)    ";
    1241: OLine2:= "O90_POSTN_SLIDE_CYL_FWD(Q1241.1)     ";
    1242: OLine2:= "O90_RH_MOVR_SUP_HORZ_CYL_FWD(Q1242.1)";
    1250: OLine2:= "O90_LH1_REJ_SLIDE_FWD(Q1250.1)       ";
    1251: OLine2:= "O90_RH2_REJ_SLIDE_FWD(Q1251.1)       ";
    1260: OLine2:= "O110_LH_OIL_SPIN_ON(Q1260.1)         ";
    1261: OLine2:= "O120_TOOL_CHO_LOCK(Q1261.1)          ";
    1262: OLine2:= "O120_CAMERA_SLIDE_CYL_FWD(Q1262.1)   ";
    ELSE
      OLine2:= " ";	
    END_CASE  
  Out_Visibility_2:=TRUE;
   
   CASE OP_Arr_OP90P[Output_Page_num] OF
    400:  Out_Lamp2:=O90_VISN_LGHT2_ON_Q400_1;
    401:  Out_Lamp2:=O90_SPARE_Q401_1;
    402:  Out_Lamp2:=O110_SPARE_Q402_1;
    403:  Out_Lamp2:=O120_TWR_LMP_GN_Q403_1;
   1240:  Out_Lamp2:=O90_RET_LH_GRIPR_CYL_OPN_Q1240_1;
   1241:  Out_Lamp2:=O90_POSTN_SLIDE_CYL_FWD_Q1241_1;
   1242:  Out_Lamp2:=O90_RH_MOVR_SUP_HORZ_CYL_FWD_Q1242_1;
   1250:  Out_Lamp2:=O90_LH1_REJ_SLIDE_FWD_Q1250_1;
   1251:  Out_Lamp2:=O90_RH2_REJ_SLIDE_FWD_Q1251_1;
   1260:  Out_Lamp2:=O110_LH_OIL_SPIN_ON_Q1260_1;
   1261:  Out_Lamp2:=O120_TOOL_CHO_LOCK_Q1261_1;
   1262:  Out_Lamp2:=O120_CAMERA_SLIDECYL_FWD_Q1262_1;
   ELSE
       Out_Visibility_2:=FALSE;	
   END_CASE 
    
    CASE OP_Arr_OP90P[Output_Page_num] OF
    400:  OLine3:= "O90_LH_DOOR_OPN(Q400.2)              ";
    401:  OLine3:= "O90_SPARE_Q401_2(Q401.2)             ";
    402:  OLine3:= "O110_SPARE_Q402_2(Q402.2)            ";
    403:  OLine3:= "O120_TWR_LMP_YELW(Q403.2)            ";
    1240: OLine3:= "O90_RET_RH_GRIPR_CYL_CLSE(Q1240.2)   ";
    1241: OLine3:= "O90_LH_MOVR_SUP_VERT_CYL_DWN(Q1241.2)";
    1242: OLine3:= "O90_SPARE_Q1242_2(Q1242.2)           ";
    1250: OLine3:= "O90_RH1_REJ_SLIDE_REV(Q1250.2)       ";
    1251: OLine3:= "O90_RH_REJ_AIR_PURGE(Q1251.2)        ";
    1260: OLine3:= "O120_RH_OIL_DISPN_ON(Q1260.2)        ";
    1261: OLine3:= "O110_PUSH_CYL_REV(Q1261.2)           ";
    1262: OLine3:= "O120_SPARE_Q1262_2(Q1262.2)          ";
    ELSE
      OLine3:= " ";	
    END_CASE
    
      Out_Visibility_3:=TRUE;	
   CASE OP_Arr_OP90P[Output_Page_num] OF
   400:  Out_Lamp3:=O90_LH_DOOR_OPN_Q400_2;
   401:  Out_Lamp3:=O90_SPARE_Q401_2;
   402:  Out_Lamp3:=O110_SPARE_Q402_2;
   403:  Out_Lamp3:=O120_TWR_LMP_YELW_Q403_2;
   1240:  Out_Lamp3:=O90_RET_RH_GRIPR_CYL_CLSE_Q1240_2;
   1241:  Out_Lamp3:=O90_LH_MOVR_SUP_VERT_CYL_DWN_Q1241_2;
   1242:  Out_Lamp3:=O90_SPARE_Q1242_2;
   1250:  Out_Lamp3:=O90_RH1_REJ_SLIDE_REV_Q1250_2;
   1251:  Out_Lamp3:=O90_RH_REJ_AIR_PURGE_Q1251_2;
   1260:  Out_Lamp3:=O110_RH_OIL_DISPN_ON_Q1260_2;
   1261:  Out_Lamp3:=O120_PUSH_CYL_REV_Q1261_2;
   1262:  Out_Lamp3:=O120_SPARE_Q1262_2;
   ELSE
       Out_Visibility_3:=FALSE;
   END_CASE 
   
    CASE OP_Arr_OP90P[Output_Page_num] OF
    400:  OLine4:= "O90_RH_DOOR_OPN(Q400.3)             ";
    401:  OLine4:= "O90_SPARE_Q401_3(Q401.3)            ";
    402:  OLine4:= "O110_SPARE_Q402_3(Q402.3)           ";
    403:  OLine4:= "O120_TWR_LMP_BUZZ(Q403.3)           ";
    1240: OLine4:= "O90_RET_RH_GRIPR_CYL_OPN(Q1240.3)   ";
    1241: OLine4:= "O90_LH_MOVR_SUP_VERT_CYL_UP(Q1241.3)";
    1242: OLine4:= "O90_SPARE_Q1242_3(Q1242.3)          ";
    1250: OLine4:= "O90_RH1_REJ_SLIDE_FWD(Q1250.3)      ";
    1251: OLine4:= "O90_SPARE_Q1251_3(Q1251.3)          ";
    1260: OLine4:= "O110_RH_OIL_SPIN_ON(Q1260.3)        ";
    1261: OLine4:= "O120_PUSH_CYL_FWD(Q1261.3)          ";
    1262: OLine4:= "O120_SPARE_Q1262_3(Q1262.3)         ";
    ELSE
      OLine4:= " ";	
    END_CASE

    Out_Visibility_4:=TRUE;
   
   CASE OP_Arr_OP90P[Output_Page_num] OF
   400:  Out_Lamp4:=O90_RH_DOOR_OPN_Q400_3;
   401:  Out_Lamp4:=O90_SPARE_Q401_3;
   402:  Out_Lamp4:=O110_SPARE_Q402_3;
   403:  Out_Lamp4:=O120_TWR_LMP_BUZZ_Q403_3;
   1240: Out_Lamp4:=O90_RET_RH_GRIPR_CYL_OPN_Q1240_3;
   1241: Out_Lamp4:=O90_LH_MOVR_SUP_VERT_CYL_UP_Q1241_3;
   1242: Out_Lamp4:=O90_SPARE_Q1242_3;
   1250: Out_Lamp4:=O90_RH1_REJ_SLIDE_FWD_Q1250_3;
   1251: Out_Lamp4:=O90_SPARE_Q1251_3;
   1260: Out_Lamp4:=O110_RH_OIL_SPIN_ON_Q1260_3;
   1261: Out_Lamp4:=O120_PUSH_CYL_FWD_Q1261_3;
   1262: Out_Lamp4:=O120_SPARE_Q1262_3;
   ELSE
       Out_Visibility_4:=FALSE;
   END_CASE 
   
    Out_Visibility_5:=TRUE;
	
    CASE OP_Arr_OP90P[Output_Page_num] OF
    400:  OLine5:= "O90_FRNT_DOOR_OPN(Q400.4)            ";
    401:  OLine5:= "O110_RH_OIL_DISPN_FRL_VLVE_ON(Q401.4) ";
    402:  OLine5:= "O120_VISN_LGHT1_ON(Q402.4)           ";
    403:  OLine5:= "O120_SPARE_Q403_4(Q403.4)            ";
    1240: OLine5:= "O90_POS_LOCK_CYL1_VLVE_1(Q1240.4)    ";
    1241: OLine5:= "O90_LH_MOVR_SUP_HORZ_CYL_REV(Q1241.4)";
    1242: OLine5:= "O90_SPARE_Q1242_4(Q1242.4)           ";
    1250: OLine5:= "O90_SPARE_Q1250_4(Q1250.4)           ";
    1251: OLine5:= "O90_SPARE_Q1251_4(Q1251.4)           ";
    1260: OLine5:= "O120_LH_GRPR_CLSE(Q1260.4)           ";
    1261: OLine5:= "O120_LH_SING_CYL_REV(Q1261.4)        ";
    1262: OLine5:= "O120_SPARE_Q1262_4(Q1262.4)          ";
    ELSE
      OLine5:= " ";	
    END_CASE
	
   CASE OP_Arr_OP90P[Output_Page_num] OF
   400:  Out_Lamp5:=O90_FRNT_DOOR_OPN_Q400_4;
   401:  Out_Lamp5:=O110_RH_OIL_DISPN_FRL_VLVE_ON_Q401_4;
   402:  Out_Lamp5:=O120_VISN_LGHT1_ON_Q402_4;
   403:  Out_Lamp5:=O120_SPARE_Q403_4;
   1240: Out_Lamp5:=O90_POS_LOCK_CYL1_VLVE_1_Q1240_4;
   1241: Out_Lamp5:=O90_LH_MOVR_SUP_HORZ_CYL_REV_Q1241_4;
   1242: Out_Lamp5:=O90_SPARE_Q1242_4;
   1250: Out_Lamp5:=O90_SPARE_Q1250_4;
   1251: Out_Lamp5:=O90_SPARE_Q1251_4;
   1260: Out_Lamp5:=O120_LH_GRPR_CLSE_Q1260_4;
   1261: Out_Lamp5:=O120_LH_SING_CYL_REV_Q1261_4;
   1262: Out_Lamp5:=O120_SPARE_Q1262_4;
   ELSE          
       Out_Visibility_5:=FALSE;
   END_CASE 
   
    Out_Visibility_6:=TRUE;

    
    CASE OP_Arr_OP90P[Output_Page_num] OF
    400:  OLine6:= "O90_BACK_DOOR_OPN(Q400.5)            ";
    401:  OLine6:= "O20_RH_OIL_DISPN_FRL_VLVE_ON(Q401.5)";
    402:  OLine6:= "O120_VISN_LGHT2_ON(Q402.5)           ";
    403:  OLine6:= "O120_SPARE_Q403_5(Q403.5)            ";
    1240: OLine6:= "O90_POS_LOCK_CYL1_VLVE_2(Q1240.5)    ";
    1241: OLine6:= "O90_LH_MOVR_SUP_HORZ_CYL_FWD(Q1241.5)";
    1242: OLine6:= "O90_SPARE_Q1242_5(Q1242.5)           ";
    1250: OLine6:= "O90_LH1_REJ_AIR_PURGE(Q1250.5)       ";
    1251: OLine6:= "O90_SPARE_Q1251_5(Q1251.5)           ";
    1260: OLine6:= "O120_LH_GRPR_OPN(Q1260.5)            ";
    1261: OLine6:= "O120_LH_SING_CYL_FWD(Q1261.5)        ";
    1262: OLine6:= "O120_SPARE_Q1262_5(Q1262.5)          ";
    ELSE
      OLine6:= " ";	
    END_CASE
		
   CASE OP_Arr_OP90P[Output_Page_num] OF
   400:  Out_Lamp6:=O90_BACK_DOOR_OPN_Q400_5;
   401:  Out_Lamp6:=O20_RH_OIL_DISPN_FRL_VLVE_ON_Q401_5;
   402:  Out_Lamp6:=O120_VISN_LGHT2_ON_Q402_5;
   403:  Out_Lamp6:=O120_SPARE_Q403_5;
   1240: Out_Lamp6:=O90_POS_LOCK_CYL1_VLVE_2_Q1240_5;
   1241: Out_Lamp6:=O90_LH_MOVR_SUP_HORZ_CYL_FWD_Q1241_5;
   1242: Out_Lamp6:=O90_SPARE_Q1242_5;
   1250: Out_Lamp6:=O90_LH1_REJ_AIR_PURGE_Q1250_5;
   1251: Out_Lamp6:=O90_SPARE_Q1251_5;
   1260: Out_Lamp6:=O120_LH_GRPR_OPN_Q1260_5;
   1261: Out_Lamp6:=O120_LH_SING_CYL_FWD_Q1261_5;
   1262: Out_Lamp6:= O120_SPARE_Q1262_5;
   ELSE          
       Out_Visibility_6:=FALSE;
   END_CASE 
    
	Out_Visibility_7:=TRUE;
    
    CASE OP_Arr_OP90P[Output_Page_num] OF
    400:  OLine7:= "O90_IPC_P_S(Q400.6)             ";
    401:  OLine7:= "O110_LH_OIL_DISPN_FRL_VLVE_ON(Q401.6) ";
    402:  OLine7:= "O120_BARLIGHT_OP1(Q402.6)            ";
    403:  OLine7:= "O120_SPARE_Q403_6(Q403.6)            ";
    1240: OLine7:= "O90_POS_LOCK_CYL2_VLVE_1(Q1240.6)    ";
    1241: OLine7:= "O90_RH_MOVR_SUP_VERT_CYL_DWN(Q1241.6)";
    1242: OLine7:= "O90_SPARE_Q1242_6(Q1242.6)           ";
    1250: OLine7:= "O90_LH2_REJ_SLIDE_REV(Q1250.6)       ";
    1251: OLine7:= "O90_SPARE_Q1251_6(Q1251.6)           ";
    1260: OLine7:= "O120_LH_REJ_AIR_PURGE(Q1260.6)       ";
    1261: OLine7:= "O120_RH_GRPR_CLSE(Q1261.6)           ";
    1262: OLine7:= "O120_SPARE_Q1262_6(Q1262.6)          ";
    ELSE
      OLine7:= " ";	
    END_CASE
    	
   CASE OP_Arr_OP90P[Output_Page_num] OF
   400:  Out_Lamp7:=O90_IPC_P_S_Q400_6;
   401:  Out_Lamp7:=O110_LH_OIL_DISPN_FRL_VLVE_ON_Q401_6;
   402:  Out_Lamp7:=O120_BARLIGHT_OP1_Q402_6;
   403:  Out_Lamp7:=O120_SPARE_Q403_6;
   1240: Out_Lamp7:=O90_POS_LOCK_CYL2_VLVE_1_Q1240_6;
   1241: Out_Lamp7:=O90_RH_MOVR_SUP_VERT_CYL_DWN_Q1241_6;
   1242: Out_Lamp7:=O90_SPARE_Q1242_6;
   1250: Out_Lamp7:=O90_LH2_REJ_SLIDE_REV_Q1250_6;
   1251: Out_Lamp7:=O90_SPARE_Q1251_6;
   1260: Out_Lamp7:=O120_RH_GRPR_CLSE_Q1260_6;
   1261: Out_Lamp7:=O120_LH_REJ_AIR_PURGE_Q1261_6;
   1262: Out_Lamp7:=O120_SPARE_Q1262_6;
   ELSE
       Out_Visibility_7:=FALSE;
   END_CASE 
   
    CASE OP_Arr_OP90P[Output_Page_num] OF
    400:  OLine8:= "O90_SPARE_Q400_7(Q400.7)            ";
    401:  OLine8:= "O20_LH_OIL_DISPN_FRL_VLVE_ON(Q401.7)";
    402:  OLine8:= "O120_BARLIGHT_OP2(Q402.7)           ";
    403:  OLine8:= "O120_SPARE_Q403_7(Q403.7)           ";
    1240: OLine8:= "O90_POS_LOCK_CYL2_VLVE_2(Q1240.7)   ";
    1241: OLine8:= "O90_RH_MOVR_SUP_VERT_CYL_UP(Q1241.7)";
    1242: OLine8:= "O90_SPARE_Q1242_7(Q1242.7)          ";
    1250: OLine8:= "O90_LH2_REJ_SLIDE_FWD(Q1250.7)      ";
    1251: OLine8:= "O90_SPARE_Q1251_7(Q1251.7)          ";
    1260: OLine8:= "O120_RH_GRPR_OPN(Q1260.7)           ";
    1261: OLine8:= "O120_RH_REJ_AIR_PURGE(Q1261.7)      ";
    1262: OLine8:= "O120_SPARE_Q1262_7(Q1262.7)         ";
    ELSE
      OLine8:= " ";	
    END_CASE
	
    Out_Visibility_8:=TRUE;
   
   CASE OP_Arr_OP90P[Output_Page_num] OF
   400:  Out_Lamp8:=O90_SPARE_Q400_7;
   401:  Out_Lamp8:=O20_LH_OIL_DISPN_FRL_VLVE_ON_Q401_7;
   402:  Out_Lamp8:=O120_BARLIGHT_OP2_Q402_7;
   403:  Out_Lamp8:=O120_SPARE_Q403_7;
   1240: Out_Lamp8:=O90_POS_LOCK_CYL2_VLVE_2_Q1240_7;
   1241: Out_Lamp8:=O90_RH_MOVR_SUP_VERT_CYL_UP_Q1241_7;
   1242: Out_Lamp8:=O90_SPARE_Q1242_7;
   1250: Out_Lamp8:=O90_LH2_REJ_SLIDE_FWD_Q1250_7;
   1251: Out_Lamp8:=O90_SPARE_Q1251_7;
   1260: Out_Lamp8:=O120_RH_GRPR_OPN_Q1260_7;
   1261: Out_Lamp8:=O120_RH_REJ_AIR_PURGE_Q1261_7;
   1262: Out_Lamp8:=O120_SPARE_Q1262_7;
   ELSE           
       Out_Visibility_8:=FALSE;	
   END_CASE   
   
 3: CASE IP_Arr_OP160P[Input_Page_num] OF
    700: Line1:= "I130_LH_ATC_DECLAMP_FB(I700.0)";
    701: Line1:= "I130_RH_ATC_DECLAMP_FB(I701.0)";
    702: Line1:= "I140_ATC1_DECLAMP_FB(I702.0)  ";
    703: Line1:= "I140_SPARE_I703_0(I703.0)     ";
    704: Line1:= "I140_SPARE_I704_0(I704.0)     ";
    705: Line1:= "I140_ATC2_DECLAMP_FB(I705.0)  ";
    706: Line1:= "I140_SPARE_I706_0(I706.0)     ";
    707: Line1:= "I140_SPARE_I707_0(I707.0)     ";
    708: Line1:= "I140_ATC3_DECLAMP_FB(I708.0)  ";
    709: Line1:= "I140_SPARE_I709_0(I709.0)     ";
    710: Line1:= "I140_SPARE_I710_0(I710.0)"     ;
    711: Line1:= "I160_ATC1_STN_POKE_YOKE_1(I711.0)" ;
    712: Line1:= "I160_RH_COMP_PP_GRPR_CLSE(I712.0)" ;
    //713: Line1:="I160_SPARE_I713_0(I713.0)" ;
    714: Line1:= "I10A_DRUM_FEED_ALRM(I714.0)" ;
    715: Line1:= "I160_SPARE_I715_0(I715.0)";
    1300:Line1:= "I130_LH_ROTRY_0_DEG(I1300.0)" ;
    1301:Line1:= "I140_HORZ_SUP1_CYL_REV(I1301.0)" ;
    1310:Line1:= "I140_HORZ_SUP2_CYL_REV(I1310.0)" ;
    1311:Line1:= "I140_VERT_SUP3_CYL_REV(I1311.0)" ;
    1320:Line1:= "I160_SLIDE_CYL_REV(I1320.0)" ;
    1321:Line1:= "I160_SPARE_I1321_0(I1321.0)" ;
    1330:Line1:= "I160_LH_PALLET_LOCK_CYL_UNLOCK(I1330.0)" ;
    1331:Line1:= "I160_REJ_BOX_DOOR_CLSE(I1331.0)";
    ELSE
      Line1:= " ";	
    END_CASE
  Visibility_1:=TRUE;
      
   CASE IP_Arr_OP160P[Input_Page_num] OF
	700: Lamp1:=I130_LH_ATC_DECLAMP_FBI700_0 ;
	701: Lamp1:=I130_RH_ATC_DECLAMP_FBI701_0 ;
	702: Lamp1:=I140_ATC1_DECLAMP_FBI702_0 ;
	703: Lamp1:=I140_SPARE_I703_0 ;
	704: Lamp1:=I140_SPARE_I704_0I704_0  ;
	705: Lamp1:=I140_ATC2_DECLAMP_FBI705_0 ;
	706: Lamp1:=I140_SPARE_I706_0 ;
	707: Lamp1:=I140_SPARE_I707_0 ;
	708: Lamp1:=I140_ATC3_DECLAMP_FBI708_0 ;
	709: Lamp1:=I140_SPARE_I709_0 ;
	710: Lamp1:=I140_SPARE_I710_0 ;
	711: Lamp1:=I160_ATC1_STN_POKE_YOKE_1I711_0 ;
	712: Lamp1:=I160_RH_COMP_PP_GRPR_CLSEI712_0 ;
	//713: Lamp1:=I160_SPARE_I713_0 ;
	714: Lamp1:=I10A_DRUM_FEED_ALRMI714_0 ;
	715: Lamp1:=I160_SPARE_I715_0 ;
	1300:Lamp1:=I130_LH_ROTRY_0_DEGI1300_0 ;
	1301:Lamp1:=I140_HORZ_SUP1_CYL_REVI1301_0 ;
	1310:Lamp1:=I140_HORZ_SUP2_CYL_REVI1310_0 ;
	1311:Lamp1:=I140_VERT_SUP3_CYL_REVI1311_0 ;
	1320:Lamp1:=I160_SLIDE_CYL_REVI1320_0 ;
	1321:Lamp1:=I160_SPARE_I1321_0 ;
	1330:Lamp1:=I160_LH_PALLET_LOCK_CYL_UNLOCKI1330_0 ;
	1331:Lamp1:=I160_REJ_BOX_DOOR_CLSEI1331_0 ;
   ELSE
       Visibility_1:=FALSE;	
   END_CASE
  
    CASE IP_Arr_OP160P[Input_Page_num] OF
    700: Line2:= "I130_LH_ATC_CLAMP_FB(I700.1)";
    701: Line2:= "I130_RH_ATC_CLAMP_FB(I701.1)";
    702: Line2:= "I140_ATC1_CLAMP_FB(I702.1)  ";
    703: Line2:= "I140_SPARE_I703_1(I703.1)   ";
    704: Line2:= "I140_LK_TST_2_PAS(I704.1)   ";
    705: Line2:= "I140_ATC2_CLAMP_FB(I705.1)  ";
    706: Line2:= "I140_LK_TST_3_PAS(I706.1)   ";
    707: Line2:= "I140_LK_TST_4_PAS(I707.1)   ";
    708: Line2:= "I140_ATC3_CLAMP_FB(I708.1)  ";
    709: Line2:= "I140_SPARE_I709_1(I709.1)   ";
    710: Line2:= "I140_LK_TST_6_PAS(I710.1)" ;
    711: Line2:= "I160_ATC1_STN_POKE_YOKE_2(I711.1)" ;
    712: Line2:= "I160_RH_COMP_PP_GRPR_OPN(I712.1)" ;
    //713: Line2:="I160_SPARE_I713_1(I713.1)" ;
    714: Line2:= "I10A_SPARE_I714_1(I714.1)" ;
    715: Line2:= "I160_SPARE_I715_1(I715.1) ";
    1300:Line2:= "I130_LH_ROTRY_180_DEG(I1300.1)" ;
    1301:Line2:= "I140_HORZ_SUP1_CYL_FWD(I1301.1)" ;
    1310:Line2:= "I140_HORZ_SUP2_CYL_FWD(I1310.1)" ;
    1311:Line2:= "I140_VERT_SUP3_CYL_FWD(I1311.1)" ;
    1320:Line2:= "I160_SLIDE_CYL_FWD(I1320.1)" ;
    1321:Line2:= "I160_SPARE_I1321_1(I1321.1)" ;
    1330:Line2:= "I160_LH_PALLET_LOCK_CYL_LOCK(I1330.1)" ;
    1331:Line2:= "I160_SAM_PART_BAG_DOOR_CLSE(I1331.1)" ;
    ELSE
      Line2:= " ";	
    END_CASE
       Visibility_2:=TRUE;

    CASE IP_Arr_OP160P[Input_Page_num] OF
	700: Lamp2:=I130_LH_ATC_CLAMP_FBI700_1 ;
	701: Lamp2:=I130_RH_ATC_CLAMP_FBI701_1 ;
	702: Lamp2:=I140_ATC1_CLAMP_FBI702_1 ;
	703: Lamp2:=I140_SPARE_I703_1 ;
	704: Lamp2:=I140_LK_TST_2_PASI704_1  ;
	705: Lamp2:=I140_ATC2_CLAMP_FBI705_1 ;
	706: Lamp2:=I140_LK_TST_3_PASI706_1 ;
	707: Lamp2:=I140_LK_TST_4_PASI707_1 ;
	708: Lamp2:=I140_ATC3_CLAMP_FBI708_1 ;
	709: Lamp2:=I140_SPARE_I709_1 ;
	710: Lamp2:=I140_LK_TST_6_PASI710_1 ;
	711: Lamp2:=I160_ATC1_STN_POKE_YOKE_2I711_1 ;
	712: Lamp2:=I160_RH_COMP_PP_GRPR_OPNI712_1 ;
	//713: Lamp2:=I160_SPARE_I713_1 ;
	714: Lamp2:=I10A_SPARE_I714_1 ;
	715: Lamp2:=I160_SPARE_I715_1 ;
	1300:Lamp2:=I130_LH_ROTRY_180_DEGI1300_1 ;
	1301:Lamp2:=I140_HORZ_SUP1_CYL_FWDI1301_1 ;
	1310:Lamp2:=I140_HORZ_SUP2_CYL_FWDI1310_1 ;
	1311:Lamp2:=I140_VERT_SUP3_CYL_FWDI1311_1 ;
	1320:Lamp2:=I160_SLIDE_CYL_FWDI1320_1 ;
	1321:Lamp2:=I160_SPARE_I1321_1 ;
	1330:Lamp2:=I160_LH_PALLET_LOCK_CYL_LOCKI1330_1 ;
	1331:Lamp2:=I160_SAM_PART_BAG_DOOR_CLSEI1331_1 ;
   ELSE
       Visibility_2:=FALSE;	
   END_CASE

    CASE IP_Arr_OP160P[Input_Page_num] OF
    700: Line3:= "I130_LH_ATC_STN_POKE_YOKE_1(I700.2)";
    701: Line3:= "I130_RH_ATC_STN_POKE_YOKE_1(I701.2)";
    702: Line3:= "I140_ATC1_STN_POKE_YOKE_1(I702.2)  ";
    703: Line3:= "I140_SPARE_I703_2(I703.2)          ";
    704: Line3:= "I140_LK_TST_2_FL(I704.2)           ";
    705: Line3:= "I140_ATC2_STN_POKE_YOKE_1(I705.2)  ";
    706: Line3:= "I140_LK_TST_3_FL(I706.2)           ";
    707: Line3:= "I140_LK_TST_4_FL(I707.2)           ";
    708: Line3:= "I140_ATC3_STN_POKE_YOKE_1(I708.2)  ";
    709: Line3:= "I140_SPARE_I709_2(I709.2)          ";
    710: Line3:= "I140_LK_TST_6_FL(I710.2)" ;
    711: Line3:= "I160_ATC1_STN_POKE_YOKE_3(I711.2)" ;
    712: Line3:= "I160_AUTOBAG_READY(I712.2)" ;
    713: Line3:= "I160_VFD_RDY(I713.2)" ;
    714: Line3:= "I10A_DRUM_OFF_ON(I714.2)" ;
    715: Line3:= "I160_SPARE_I715_2(I715.2)" ;
    1300:Line3:= "I130_RH_ROTRY_0_DEG(I1300.2)" ;
    1301:Line3:= "I140_VERT_SUP1_CYL_REV(I1301.2)" ;
    1310:Line3:= "I140_VERT_SUP2_CYL_REV(I1310.2)" ;
    1311:Line3:= "I140_WIPE3_CYL_REV(I1311.2)" ;
    1320:Line3:= "I160_SLAVE1_PRSN_PARK_TRAY(I1320.2)" ;
    1321:Line3:= "I160_SPARE_I1321_2(I1321.2)";
    1330:Line3:= "I160_RH_PALLET_LOCK_CYL_UNLOCK(I1330.2)" ;
    1331:Line3:= "I160_TROLLEY_FIXT_PRSN(I1331.2)" ; 
    ELSE
      Line3:= " ";	
    END_CASE
       Visibility_3:=TRUE;

   CASE IP_Arr_OP160P[Input_Page_num] OF
	700: Lamp3:=I130_LH_ATC_STN_POKE_YOKE_1I700_2 ;
	701: Lamp3:=I130_RH_ATC_STN_POKE_YOKE_1I701_2 ;
	702: Lamp3:=I140_ATC1_STN_POKE_YOKE_1I702_2 ;
	703: Lamp3:=I140_SPARE_I703_2 ;
	704: Lamp3:=I140_LK_TST_2_FLI704_2  ;
	705: Lamp3:=I140_ATC2_STN_POKE_YOKE_1I705_2 ;
	706: Lamp3:=I140_LK_TST_3_FLI706_2 ;
	707: Lamp3:=I140_LK_TST_4_FLI707_2 ;
	708: Lamp3:=I140_ATC3_STN_POKE_YOKE_1I708_2 ;
	709: Lamp3:=I140_SPARE_I709_2 ;
	710: Lamp3:=I140_LK_TST_6_FLI710_2 ;
	711: Lamp3:=I160_ATC1_STN_POKE_YOKE_3I711_2 ;
	712: Lamp3:=I160_AUTOBAG_READYI712_2 ;
	713: Lamp3:=I160_VFD_RDYI713_2 ;
	714: Lamp3:=I10A_DRUM_OFF_ON_I714_2 ;
	715: Lamp3:=I160_SPARE_I715_2 ;
	1300:Lamp3:=I130_RH_ROTRY_0_DEGI1300_2 ;
	1301:Lamp3:=I140_VERT_SUP1_CYL_REVI1301_2 ;
	1310:Lamp3:=I140_VERT_SUP2_CYL_REVI1310_2 ;
	1311:Lamp3:=I140_WIPE3_CYL_REVI1311_2 ;
	1320:Lamp3:=I160_SLAVE1_PRSN_PARK_TRAYI1320_2 ;
	1321:Lamp3:=I160_SPARE_I1321_2 ;
	1330:Lamp3:=I160_RH_PALLET_LOCK_CYL_UNLOCKI1330_2 ;
	1331:Lamp3:=I160_TROLLEY_FIXT_PRSNI1331_2 ;
   ELSE
       Visibility_3:=FALSE;	
   END_CASE

    CASE IP_Arr_OP160P[Input_Page_num] OF
    700: Line4:= "I130_LH_ATC_STN_POKE_YOKE_2(I700.3)";
    701: Line4:= "I130_RH_ATC_STN_POKE_YOKE_2(I701.3)";
    702: Line4:= "I140_ATC1_STN_POKE_YOKE_2(I702.3)  ";
    703: Line4:= "I140_LK_TST_1_PAS(I703.3)          ";
    704: Line4:= "I140_LK_TST_2_REF_PRT_FL(I704.3)   ";
    705: Line4:= "I140_ATC2_STN_POKE_YOKE_2(I705.3)  ";
    706: Line4:= "I140_LK_TST_3_REF_PRT_FL(I706.3)   ";
    707: Line4:= "I140_LK_TST_4_REF_PRT_FL(I707.3)   ";
    708: Line4:= "I140_ATC3_STN_POKE_YOKE_2(I708.3)  ";
    709: Line4:= "I140_LK_TST_5_PAS(I709.3)          ";
    710: Line4:= "I140_LK_TST_6_REF_PRT_FL(I710.3)"   ;
    711: Line4:= "I160_ATC1_STN_POKE_YOKE_4(I711.3)"  ;
    //712: Line4:="I160_SPARE_I712_3(I712.3)"         ;
    713: Line4:= "I160_SPARE_I713_3(I713.3)"          ;
    714: Line4:= "I10A_DRUM_CONV_REV(I714.3)"         ;
    715: Line4:= "I160_SPARE_I715_3(I715.3)"          ;
    1300:Line4:= "I130_RH_ROTRY_180_DEG(I1300.3)"     ;
    1301:Line4:= "I140_VERT_SUP1_CYL_FWD(I1301.3)"    ;
    1310:Line4:= "I140_VERT_SUP2_CYL_FWD(I1310.3)"    ;
    1311:Line4:= "I140_WIPE3_CYL_FWD(I1311.3)"        ;
    1320:Line4:= "I160_SLAVE2_PRSN_PARK_TRAY(I1320.3)" ;
    1321:Line4:= "I160_SPARE_I1321_3(I1321.3)"        ;
    1330:Line4:= "I160_RH_PALLET_LOCK_CYL_LOCK(I1330.3)" ;
    1331:Line4:= "I160_SAM_BOX_DOOR_CLSE(I1331.3)"    ;
    ELSE
      Line4:= " ";	
    END_CASE
       Visibility_4:=TRUE;
   
   CASE IP_Arr_OP160P[Input_Page_num] OF
	700: Lamp4:=I130_LH_ATC_STN_POKE_YOKE_2I700_3 ;
	701: Lamp4:=I130_RH_ATC_STN_POKE_YOKE_2I701_3 ;
	702: Lamp4:=I140_ATC1_STN_POKE_YOKE_2I702_3 ;
	703: Lamp4:=I140_LK_TST_1_PASI703_3 ;
	704: Lamp4:=I140_LK_TST_2_REF_PRT_FLI704_3  ;
	705: Lamp4:=I140_ATC2_STN_POKE_YOKE_2I705_3 ;
	706: Lamp4:=I140_LK_TST_3_REF_PRT_FLI706_3 ;
	707: Lamp4:=I140_LK_TST_4_REF_PRT_FLI707_3 ;
	708: Lamp4:=I140_ATC3_STN_POKE_YOKE_2I708_3 ;
	709: Lamp4:=I140_LK_TST_5_PASI709_3 ;
	710: Lamp4:=I140_LK_TST_6_REF_PRT_FLI710_3 ;
	711: Lamp4:=I160_ATC1_STN_POKE_YOKE_4I711_3 ;
	//712: Lamp4:=I160_SPARE_I712_3 ;
	713: Lamp4:=I160_SPARE_I713_3 ;
	714: Lamp4:=I10A_DRUM_CONV_REV_I714_3 ;
	715: Lamp4:=I160_SPARE_I715_3 ;
	1300:Lamp4:=I130_RH_ROTRY_180_DEGI1300_3 ;
	1301:Lamp4:=I140_VERT_SUP1_CYL_FWDI1301_3 ;
	1310:Lamp4:=I140_VERT_SUP2_CYL_FWDI1310_3 ;
	1311:Lamp4:=I140_WIPE3_CYL_FWDI1311_3 ;
	1320:Lamp4:=I160_SLAVE2_PRSN_PARK_TRAYI1320_3 ;
	1321:Lamp4:=I160_SPARE_I1321_3 ;
	1330:Lamp4:=I160_RH_PALLET_LOCK_CYL_LOCKI1330_3 ;
	1331:Lamp4:=I160_SAM_BOX_DOOR_CLSEI1331_3 ;
   ELSE
       Visibility_4:=FALSE;	
   END_CASE
    
    CASE IP_Arr_OP160P[Input_Page_num] OF
    700: Line5:= "I130_LH_ATC_STN_POKE_YOKE_3(I700.4)";
    701: Line5:= "I130_RH_ATC_STN_POKE_YOKE_3(I701.4)";
    702: Line5:= "I140_ATC1_STN_POKE_YOKE_3(I702.4)  ";
    703: Line5:= "I140_LK_TST_1_FL(I703.4)           ";
    704: Line5:= "I140_LK_TST_2_WARNG(I704.4)        ";
    705: Line5:= "I140_ATC2_STN_POKE_YOKE_3(I705.4)  ";
    706: Line5:= "I140_LK_TST_3_WARNG(I706.4)        ";
    707: Line5:= "I140_LK_TST_4_WARNG(I707.4)        ";
    708: Line5:= "I140_ATC3_STN_POKE_YOKE_3(I708.4)  ";
    709: Line5:= "I140_LK_TST_5_FL(I709.4)           ";
    710: Line5:= "I140_LK_TST_6_WARNG(I710.4)" ;
    711: Line5:= "I160_ATC1_SLAVE_TOOL1(I711.4)" ;
    //712: Line5:="I160_SPARE_I712_4(I712.4)" ;
    713: Line5:= "I160_SPARE_I713_4(I713.4)" ;
    714: Line5:= "I10A_DRUM_CONV_FWD(I714.4)" ;
    715: Line5:= "I160_SPARE_I715_4(I715.4)" ;
    //1300:Line5:="I130_SPARE_I1300_4(I1300.4)" ;
    1301:Line5:= "I140_WIPE1_CYL_REV(I1301.4)" ;
    1310:Line5:= "I140_WIPE2_CYL_REV(I1310.4)" ;
    1311:Line5:= "I140_LEAKTEST_PRESS_SW(I1311.4)" ;
    1320:Line5:= "I160_FIXT_COMP1_PRSN(I1320.4)" ;
    1321:Line5:= "I160_SPARE_I1321_4(I1321.4)" ;
    1330:Line5:= "I160_SPARE_I1330_4(I1330.4)" ;
    1331:Line5:= "I160_SPARE_I1331_4(I1331.4)" ;
    ELSE
      Line5:= " ";	
    END_CASE
       Visibility_5:=TRUE;
   
   CASE IP_Arr_OP160P[Input_Page_num] OF
	700: Lamp5:=I130_LH_ATC_STN_POKE_YOKE_3I700_4 ;
	701: Lamp5:=I130_RH_ATC_STN_POKE_YOKE_3I701_4 ;
	702: Lamp5:=I140_ATC1_STN_POKE_YOKE_3I702_4 ;
	703: Lamp5:=I140_LK_TST_1_FLI703_4 ;
	704: Lamp5:=I140_LK_TST_2_WARNGI704_4  ;
	705: Lamp5:=I140_ATC2_STN_POKE_YOKE_3I705_4 ;
	706: Lamp5:=I140_LK_TST_3_WARNGI706_4 ;
	707: Lamp5:=I140_LK_TST_4_WARNGI707_4 ;
	708: Lamp5:=I140_ATC3_STN_POKE_YOKE_3I708_4 ;
	709: Lamp5:=I140_LK_TST_5_FLI709_4 ;
	710: Lamp5:=I140_LK_TST_6_WARNGI710_4 ;
	711: Lamp5:=I160_ATC1_SLAVE_TOOL1I711_4 ;
	//712: Lamp5:=I160_SPARE_I712_4 ;
	713: Lamp5:=I160_SPARE_I713_4 ;
	714: Lamp5:=I10A_DRUM_CONV_FWD_I714_4 ;
	715: Lamp5:=I160_SPARE_I715_4 ;
	//1300:Lamp5:=I130_SPARE_I1300_4 ;
	1301:Lamp5:=I140_WIPE1_CYL_REVI1301_4 ;
	1310:Lamp5:=I140_WIPE2_CYL_REVI1310_4 ;
	1311:Lamp5:=I140_LEAKTEST_PRESS_SWI1311_4 ;
	1320:Lamp5:=I160_FIXT_COMP1_PRSNI1320_4 ;
	1321:Lamp5:=I160_SPARE_I1321_4 ;
	1330:Lamp5:=I160_SPARE_I1330_4 ;
	1331:Lamp5:=I160_SPARE_I1331_4 ;
   ELSE
       Visibility_5:=FALSE;	
   END_CASE
   
    CASE IP_Arr_OP160P[Input_Page_num] OF
    700: Line6:= "I130_LH_ATC_STN_POKE_YOKE_4(I700.5)";
    701: Line6:= "I130_RH_ATC_STN_POKE_YOKE_4(I701.5)";
    702: Line6:= "I140_ATC1_STN_POKE_YOKE_4(I702.5)  ";
    703: Line6:= "I140_LK_TST_1_REF_PRT_FL(I703.5)   ";
    704: Line6:= "I140_LK_TST_2_END_CYC(I704.5)      ";
    705: Line6:= "I140_ATC2_STN_POKE_YOKE_4(I705.5)  ";
    706: Line6:= "I140_LK_TST_3_END_CYC(I706.5)      ";
    707: Line6:= "I140_LK_TST_4_END_CYC(I707.5)      ";
    708: Line6:= "I140_ATC3_STN_POKE_YOKE_4(I708.5)  ";
    709: Line6:= "I140_LK_TST_5_REF_PRT_FL(I709.5)   ";
    710: Line6:= "I140_LK_TST_6_END_CYC(I710.5)" ;
    711: Line6:= "I160_ATC1_SLAVE_TOOL2(I711.5)" ;
    712: Line6:= "I160_AUTOBAG_ERR_STOP(I712.5)" ;
    713: Line6:= "I160_SPARE_I713_5(I713.5)";
    714: Line6:= "I10A_ROB_MAN_AUTO_MODE(I714.5)" ;
    715: Line6:= "I160_SPARE_I715_5(I715.5)" ;
    //1300:Line6:="I130_SPARE_I1300_5(I1300.5)" ;
    1301:Line6:= "I140_WIPE1_CYL_FWD(I1301.5)" ;
    1310:Line6:= "I140_WIPE2_CYL_FWD(I1310.5)" ;
    1311:Line6:= "I140_SPARE_I1311_5(I1311.5)" ;
    1320:Line6:= "I160_FIXT_COMP2_PRSN(I1320.5)" ;
    1321:Line6:= "I160_SPARE_I1321_5(I1321.5)" ;
    1330:Line6:= "I160_CONV_BDY_PRSN1_SEN(I1330.5)" ;
    1331:Line6:= "I160_SPARE_I1331_5(I1321.5)" ;
    ELSE
      Line6:= " ";	
    END_CASE   
       Visibility_6:=TRUE;
   
   CASE IP_Arr_OP160P[Input_Page_num] OF
	700: Lamp6:=I130_LH_ATC_STN_POKE_YOKE_4I700_5 ;
	701: Lamp6:=I130_RH_ATC_STN_POKE_YOKE_4I701_5 ;
	702: Lamp6:=I140_ATC1_STN_POKE_YOKE_4I702_5 ;
	703: Lamp6:=I140_LK_TST_1_REF_PRT_FLI703_5 ;
	704: Lamp6:=I140_LK_TST_2_END_CYCI704_5  ;
	705: Lamp6:=I140_ATC2_STN_POKE_YOKE_4I705_5 ;
	706: Lamp6:=I140_LK_TST_3_END_CYCI706_5 ;
	707: Lamp6:=I140_LK_TST_4_END_CYCI707_5 ;
	708: Lamp6:=I140_ATC3_STN_POKE_YOKE_4I708_5 ;
	709: Lamp6:=I140_LK_TST_5_REF_PRT_FLI709_5 ;
	710: Lamp6:=I140_LK_TST_6_END_CYCI710_5 ;
	711: Lamp6:=I160_ATC1_SLAVE_TOOL2I711_5 ;
	712: Lamp6:=I160_AUTOBAG_ERR_STOPI712_5 ;
	713: Lamp6:=I160_SPARE_I713_5 ;
	714: Lamp6:=I10A_ROB_MAN_AUTO_MODE_I714_5 ;
	715: Lamp6:=I160_SPARE_I715_5 ;
	//1300:Lamp6:=I130_SPARE_I1300_5 ;
	1301:Lamp6:=I140_WIPE1_CYL_FWDI1301_5 ;
	1310:Lamp6:=I140_WIPE2_CYL_FWDI1310_5 ;
	1311:Lamp6:=I140_SPARE_I1311_5 ;
	1320:Lamp6:=I160_FIXT_COMP2_PRSNI1320_5 ;
	1321:Lamp6:=I160_SPARE_I1321_5 ;
	1330:Lamp6:=I160_CONV_BDY_PRSN1_SENI1330_5 ;
	1331:Lamp6:=I160_SPARE_I1331_5 ;
   ELSE
       Visibility_6:=FALSE;	
   END_CASE
   
    CASE IP_Arr_OP160P[Input_Page_num] OF
    700: Line7:= "I130_LH_ATC_SLAVE_MODL1(I700.6)";
    701: Line7:= "I130_RH_ATC_SLAVE_MODL1(I701.6)";
    702: Line7:= "I140_ATC1_SLAVE_MODL1(I702.6)  ";
    703: Line7:= "I140_LK_TST_1_WARNG(I703.6)    ";
    704: Line7:= "I140_SPARE_I704_6(I704.6)      ";
    705: Line7:= "I140_ATC2_SLAVE_MODL1(I705.6)  ";
    706: Line7:= "I140_SPARE_I706_6(I706.6)      ";
    707: Line7:= "I140_SPARE_I707_6(I707.6)      ";
    708: Line7:= "I140_ATC3_SLAVE_MODL1(I708.6)  ";
    709: Line7:= "I140_LK_TST_5_WARNG(I709.6)    ";
    710: Line7:= "I160_ATC_DECLAMP_FB(I710.6)" ;
    711: Line7:= "I160_FIXT_LH_COMP_PP_GRPR_CLSE(I711.6)" ;
    712: Line7:= "I20_RESRVR_LW_LVL(I712.6)" ;
    713: Line7:= "I160_SPARE_I713_6(I713.6)" ;
    714: Line7:= "I160_SPARE_I714_6(I714.6)" ;
    715: Line7:= "I160_SPARE_I715_6(I715.6)" ;
    //1300:Line7:="I130_SPARE_I1300_6(I1300.6)" ;
    1301:Line7:= "I140_SPARE_I1301_6(I1301.6)" ;
    1310:Line7:= "I140_HORZ_SUP3_CYL_REV(I1310_6)" ;
    1311:Line7:= "I160_MOVR_REM_CYL_REV(I1311_6)" ;
    1320:Line7:= "I160_SPARE_I1320_6(I1320.6)" ;
    1321:Line7:= "I160_SPARE_I1321_6(I1321.6)" ;
    1330:Line7:= "I160_CONV_BDY_PRSN2_SEN(I1330_6)" ;
    1331:Line7:= "I160_SPARE_I1331_6(I1331.6)" ;
    ELSE
      Line7:= " ";	
    END_CASE
       Visibility_7:=TRUE;
   
   CASE IP_Arr_OP160P[Input_Page_num] OF
	700: Lamp7:=I130_LH_ATC_SLAVE_MODL1I700_6 ;
	701: Lamp7:=I130_RH_ATC_SLAVE_MODL1I701_6 ;
	702: Lamp7:=I140_ATC1_SLAVE_MODL1I702_6 ;
	703: Lamp7:=I140_LK_TST_1_WARNGI703_6 ;
	704: Lamp7:=I140_SPARE_I704_6  ;
	705: Lamp7:=I140_ATC2_SLAVE_MODL1I705_6 ;
	706: Lamp7:=I140_SPARE_I706_6 ;
	707: Lamp7:=I140_SPARE_I707_6 ;
	708: Lamp7:=I140_ATC3_SLAVE_MODL1I708_6 ;
	709: Lamp7:=I140_LK_TST_5_WARNGI709_6 ;
	710: Lamp7:=I160_ATC_DECLAMP_FBI710_6 ;
	711: Lamp7:=I160_FIXT_LH_COMP_PP_GRPR_CLSEI711_6 ;
	712: Lamp7:=I20_RESRVR_LW_LVLI712_6 ;
	713: Lamp7:=I160_SPARE_I713_6 ;
	714: Lamp7:=I160_SPARE_I714_6 ;
	715: Lamp7:=I160_SPARE_I715_6 ;
	//1300:Lamp7:=I130_SPARE_I1300_6 ;
	1301:Lamp7:=I140_SPARE_I1301_6 ;
	1310:Lamp7:=I140_HORZ_SUP3_CYL_REVI1310_6 ;
	1311:Lamp7:=I160_MOVR_REM_CYL_REVI1311_6 ;
	1320:Lamp7:=I160_SPARE_I1320_6 ;
	1321:Lamp7:=I160_SPARE_I1321_6 ;
	1330:Lamp7:=I160_CONV_BDY_PRSN2_SENI1330_6 ;
	1331:Lamp7:=I160_SPARE_I1331_6 ;
   ELSE
       Visibility_7:=FALSE;	
   END_CASE
    
    CASE IP_Arr_OP160P[Input_Page_num] OF
    700: Line8:= "I130_LH_ATC_SLAVE_MODL2(I700.7)";
    701: Line8:= "I130_RH_ATC_SLAVE_MODL2(I701.7)";
    702: Line8:= "I140_ATC1_SLAVE_MODL2(I702.7)  ";
    703: Line8:= "I140_LK_TST_1_END_CYC(I703.7)  ";
    704: Line8:= "I140_SPARE_I704.7(I704.7)      ";
    705: Line8:= "I140_ATC2_SLAVE_MODL2(I705.7)  ";
    706: Line8:= "I140_SPARE_I706.7(I706.7)      ";
    707: Line8:= "I140_SPARE_I707.7(I707.7)      ";
    708: Line8:= "I140_ATC3_SLAVE_MODL2(I708.7)  ";
    709: Line8:= "I140_LK_TST_5_END_CYC(I709.7)  ";
    710: Line8:= "I160_ATC_CLAMP_FB(I710.7)" ;
    711: Line8:= "I160_FIXT_LH_COMP_PP_GRPR_OPN(I711.7)" ;
    712: Line8:= "I20_OILTANK_PRES_SW_FB(I712.7)" ;
    713: Line8:= "I160_SPARE_I713_7(I713.7)" ;
    714: Line8:= "I160_SPARE_I714_7(I714.7)" ;
    715: Line8:= "I160_SPARE_I715_7(I715.7)" ;
    //1300:Line8:="I130_SPARE_I1300_7(I1300.7)" ;
    1301:Line8:= "I140_SPARE_I1301_7(I1301.7)" ;
    1310:Line8:= "I140_HORZ_SUP3_CYL_FWD(I1310.7)" ;
    1311:Line8:= "I160_MOVR_REM_CYL_FWD(I1311.7)" ;
    1320:Line8:= "I160_SPARE_I1320_7(I1320.7)" ;
    1321:Line8:= "I160_SPARE_I1321_7(I1321.7)" ;
    1330:Line8:= "I160_SPARE_I1330_7(I1330.7)" ;
    1331:Line8:= "I160_SPARE_I1331_7(I1331.7)" ;
    ELSE
      Line8:= " ";	
    END_CASE
       Visibility_8:=TRUE;
   
   CASE IP_Arr_OP160P[Input_Page_num] OF
	700: Lamp8:=I130_LH_ATC_SLAVE_MODL2I700_7 ;
	701: Lamp8:=I130_RH_ATC_SLAVE_MODL2I701_7 ;
	702: Lamp8:=I140_ATC1_SLAVE_MODL2I702_7 ;
	703: Lamp8:=I140_LK_TST_1_END_CYCI703_7 ;
	704: Lamp8:=I140_SPARE_I704_7  ;
	705: Lamp8:=I140_ATC2_SLAVE_MODL2I705_7 ;
	706: Lamp8:=I140_SPARE_I706_7 ;
	707: Lamp8:=I140_SPARE_I707_7 ;
	708: Lamp8:=I140_ATC3_SLAVE_MODL2I708_7 ;
	709: Lamp8:=I140_LK_TST_5_END_CYCI709_7 ;
	710: Lamp8:=I160_ATC_CLAMP_FBI710_7 ;
	711: Lamp8:=I160_FIXT_LH_COMP_PP_GRPR_OPNI711_7 ;
	712: Lamp8:=I20_OILTANK_PRES_SW_FBI712_7 ;
	713: Lamp8:=I160_SPARE_I713_7 ;
	714: Lamp8:=I160_SPARE_I714_7 ;
	715: Lamp8:=I160_SPARE_I715_7 ;
	//1300:Lamp8:=I130_SPARE_I1300_7 ;
	1301:Lamp8:=I140_SPARE_I1301_7 ;
	1310:Lamp8:=I140_HORZ_SUP3_CYL_FWDI1310_7 ;
	1311:Lamp8:=I160_MOVR_REM_CYL_FWDI1311_7 ;
	1320:Lamp8:=I160_SPARE_I1320_7 ;
	1321:Lamp8:=I160_SPARE_I1321_7 ;
	1330:Lamp8:=I160_SPARE_I1330_7 ;
	1331:Lamp8:=I160_SPARE_I1331_7 ;
   ELSE
       Visibility_8:=FALSE;	
   END_CASE
 
    CASE OP_Arr_OP160P[Output_Page_num] OF
    700: OLine1:= "O140_LK_TST1 _RST(Q700.0)  "; 
    701: OLine1:= "O140_LK_TST1 _SEL7(Q701.0) ";
    702: OLine1:= "O140_LK_TST2 _SEL6(Q702.0) ";
    703: OLine1:= "O140_LK_TST3 _SEL5(Q703.0) ";
    704: OLine1:= "O140_LK_TST4 _SEL4(Q704.0) ";
    705: OLine1:= "O140_LK_TST5 _SEL3(Q705.0) ";
    706: OLine1:= "O140_LK_TST6 _SEL2(Q706.0) ";
    707: OLine1:= "O150_BARLIGHT_OP2(Q707.0)  ";
    708: OLine1:= "O160_VFD_FWD(Q708.0)       ";
    709: OLine1:= "O10A_DRUM_RUN_IND(Q709.0)  ";
    1340: OLine1:= "O130_LH_ROTRY_0_DEG(Q1340.0)";
    1341: OLine1:= "O140_HORZ_SUP1_CYL_REV(Q1341.0)";
    1342: OLine1:= "O140_HORZ_SUP2_CYL_REV(Q1342.0)";
    1343: OLine1:= "O140_HORZ_SUP3_CYL_REV(Q1343.0)";
    1350: OLine1:= "O160_VISN_CHECK_AIR_PURGE(Q1350.0)";
    1351: OLine1:= "O160_TOOL_CHO_UNLOCK(Q1351.0)";
    1352: OLine1:= "O160_SPARE_Q1352_0(Q1352.0)";
    1353: OLine1:= "O160_SPARE_Q1353_0(Q1353.0)";
    ELSE
      OLine1:= " ";	
    END_CASE
       Out_Visibility_1:=TRUE;
   
   CASE OP_Arr_OP160P[Output_Page_num] OF
	700:  Out_Lamp1:=O140_LK_TST1_RST_Q700_0;
	701:  Out_Lamp1:=O140_LK_TST1_SEL7_Q701_0;
	702:  Out_Lamp1:=O140_LK_TST2_SEL6_Q702_0;
	703:  Out_Lamp1:=O140_LK_TST3_SEL5_Q703_0;
	704:  Out_Lamp1:=O140_LK_TST4_SEL4_Q704_0;
	705:  Out_Lamp1:=O140_LK_TST5_SEL3_Q705_0;
	706:  Out_Lamp1:=O140_LK_TST6_SEL2_Q706_0;
	707:  Out_Lamp1:=O150_BARLIGHT_OP2_Q707_0;
	708:  Out_Lamp1:=O160_VFD_FWD_Q708_0;
	709:  Out_Lamp1:=O10A_DRUM_RUN_IND_Q709_0;
	1340:  Out_Lamp1:=O130_LH_ROTRY_0_DEG_Q1340_0;
	1341:  Out_Lamp1:=O140_HORZ_SUP1_CYL_REV_Q1341_0;
	1342:  Out_Lamp1:=O140_HORZ_SUP2_CYL_REV_Q1342_0;
	1343:  Out_Lamp1:=O140_HORZ_SUP3_CYL_REV_Q1343_0;
	1350:  Out_Lamp1:=O160_VISN_CHECK_AIR_PURGE_Q1350_0;
	1351:  Out_Lamp1:=O160_TOOL_CHO_UNLOCK_Q1351_0;
	1352:  Out_Lamp1:=O160_SPARE_Q1352_0;
	1353:  Out_Lamp1:=O160_SPARE_Q1353_0;
   ELSE
       Out_Visibility_1:=FALSE;	
   END_CASE
    
    CASE OP_Arr_OP160P[Output_Page_num] OF
    700: OLine2:= "O140_LK_TST1 _STRT(Q700.1)  ";
    701: OLine2:= "O140_LK_TST2 _RST(Q701.1)   ";
    702: OLine2:= "O140_LK_TST2 _SEL7(Q702.1)  ";
    703: OLine2:= "O140_LK_TST3 _SEL6(Q703.1)  ";
    704: OLine2:= "O140_LK_TST4 _SEL5(Q704.1)  ";
    705: OLine2:= "O140_LK_TST5 _SEL4(Q705.1)  ";
    706: OLine2:= "O140_LK_TST6 _SEL3(Q706.1)  ";
    707: OLine2:= "O160_CHECKER_LGHT_ON(Q707.1)";
    708: OLine2:= "O160_VFD_REV(Q708.1)        ";
    709: OLine2:= "O160_SPARE_Q709.1(Q709.1)   ";
   1340: OLine2:= "O130_LH_ROTRY_180_DEG(Q1340.1)";
   1341: OLine2:= "O140_HORZ_SUP1_CYL_FWD(Q1341.1)";
   1342: OLine2:= "O140_HORZ_SUP2_CYL_FWD(Q1342.1)";
   1343: OLine2:= "O140_HORZ_SUP3_CYL_FWD(Q1343.1)";
   1350: OLine2:= "O160_FIXT_PP_GRPR_CLSE_OPN(Q1350.1)";
   1351: OLine2:= "O160_TOOL_CHO_LOCK(Q1351.1)";
   1352: OLine2:= "O160_SPARE_Q1352_1(Q1352.1)";
   1353: OLine2:= "O160_SPARE_Q1353_1(Q1353.1)";
    ELSE
      OLine2:= " ";	
    END_CASE
       Out_Visibility_2:=TRUE;
   
   CASE OP_Arr_OP160P[Output_Page_num] OF
	700:  Out_Lamp2:=O140_LK_TST1_STRT_Q700_1;
	701:  Out_Lamp2:=O140_LK_TST2_RST_Q701_1;
	702:  Out_Lamp2:=O140_LK_TST2_SEL7_Q702_1;
	703:  Out_Lamp2:=O140_LK_TST3_SEL6_Q703_1;
	704:  Out_Lamp2:=O140_LK_TST4_SEL5_Q704_1;
	705:  Out_Lamp2:=O140_LK_TST5_SEL4_Q705_1;
	706:  Out_Lamp2:=O140_LK_TST6_SEL3_Q706_1;
	707:  Out_Lamp2:=O160_CHECKER_LGHT_ON_Q707_1;
	708:  Out_Lamp2:=O160_VFD_REV_Q708_1;
	709:  Out_Lamp2:=O160_SPARE_Q709_1_Q709_1;
        1340:  Out_Lamp2:=O130_LH_ROTRY_180_DEG_Q1340_1;
	1341:  Out_Lamp2:=O140_HORZ_SUP1_CYL_FWD_Q1341_1;
	1342:  Out_Lamp2:=O140_HORZ_SUP2_CYL_FWD_Q1342_1;
	1343:  Out_Lamp2:=O140_HORZ_SUP3_CYL_FWD_Q1343_1;
	1350:  Out_Lamp2:=O160_FIXT_PP_GRPR_CLSE_OPN_Q1350_1;
	1351:  Out_Lamp2:=O160_TOOL_CHO_LOCK_Q1351_1;
	1352:  Out_Lamp2:=O160_SPARE_Q1352_1;
	1353:  Out_Lamp2:=O160_SPARE_Q1353_1;
   ELSE
       Out_Visibility_2:=FALSE;	
   END_CASE 

    CASE OP_Arr_OP160P[Output_Page_num] OF
    700: OLine3:= "O140_LK_TST1 _SEL1(Q700.2)    ";
    701: OLine3:= "O140_LK_TST2 _STRT(Q701.2)    ";
    702: OLine3:= "O140_LK_TST3 _RST(Q702.2)     ";
    703: OLine3:= "O140_LK_TST3 _SEL7(Q703.2)    ";
    704: OLine3:= "O140_LK_TST4 _SEL6(Q704.2)    ";
    705: OLine3:= "O140_LK_TST5 _SEL5(Q705.2)    ";
    706: OLine3:= "O140_LK_TST6 _SEL4(Q706.2)    ";
    707: OLine3:= "O160_FUME_EXTRTR_ON(Q707.2)   ";
    708: OLine3:= "O160_VFD_STOP(Q708.2)         ";
    709: OLine3:= "O10A_ROB_MAN_AUTO_MODE(Q709.2)";
   1340: OLine3:= "O130_RH_ROTRY_0_DEG(Q1340.2)";
   1341: OLine3:= "O140_VERT_SUP1_CYL_REV(Q1341.2)";
   1342: OLine3:= "O140_VERT_SUP2_CYL_REV(Q1342.2)";
   1343: OLine3:= "O140_VERT_SUP3_CYL_REV(Q1343.2)";
   1350: OLine3:= "O160_LH_COMP_PP_GRPR_CLSE_OPN(Q1350.2)";
   1351: OLine3:= "O160_LH_PALLET_LOCK_CYL_UNLOCK(Q1351.2)";
   1352: OLine3:= "OP160_MOVR_REM_CYL_REV(Q1352.2)";
   1353: OLine3:= "O160_SPARE_Q1353_2(Q1353.2)";
    ELSE
      OLine3:= " ";	
    END_CASE
       Out_Visibility_3:=TRUE;
	
   CASE OP_Arr_OP160P[Output_Page_num] OF
	700:  Out_Lamp3:=O140_LK_TST1_SEL1_Q700_2;
	701:  Out_Lamp3:=O140_LK_TST2_STRT_Q701_2;
	702:  Out_Lamp3:=O140_LK_TST3_RST_Q702_2;
	703:  Out_Lamp3:=O140_LK_TST3_SEL7_Q703_2;
	704:  Out_Lamp3:=O140_LK_TST4_SEL6_Q704_2;
	705:  Out_Lamp3:=O140_LK_TST5_SEL5_Q705_2;
	706:  Out_Lamp3:=O140_LK_TST6_SEL4_Q706_2;
	707:  Out_Lamp3:=O160_FUME_EXTRTR_ON_Q707_2;
	708:  Out_Lamp3:=O160_VFD_STOP_Q708_2;
	709:  Out_Lamp3:=O10A_ROB_MAN_AUTO_MODE_Q709_2;
   1340:  Out_Lamp3:=O130_RH_ROTRY_0_DEG_Q1340_2;
	1341:  Out_Lamp3:=O140_VERT_SUP1_CYL_REV_Q1341_2;
	1342:  Out_Lamp3:=O140_VERT_SUP2_CYL_REV_Q1342_2;
	1343:  Out_Lamp3:=O140_VERT_SUP3_CYL_REV_Q1343_2;
	1350:  Out_Lamp3:=O160_LH_COMP_PP_GRPR_CLSE_OPN_Q1350_2;
	1351:  Out_Lamp3:=O160_LH_PALLET_LOCK_CYL_UNLOCK_Q1351_2;
	1352:  Out_Lamp3:=OP160_MOVR_REM_CYL_REV_Q1352_2;
	1353:  Out_Lamp3:=O160_SPARE_Q1353_2;
   ELSE
       Out_Visibility_3:=FALSE;
   END_CASE 
    
    CASE OP_Arr_OP160P[Output_Page_num] OF
    700: OLine4:= "O140_LK_TST1 _SEL2(Q700.3)    ";
    701: OLine4:= "O140_LK_TST2 _SEL1(Q701.3)    ";
    702: OLine4:= "O140_LK_TST3 _STRT(Q702.3)    ";
    703: OLine4:= "O140_LK_TST4 _RST(Q703.3)     ";
    704: OLine4:= "O140_LK_TST4 _SEL7(Q704.3)    ";
    705: OLine4:= "O140_LK_TST5 _SEL6(Q705.3)    ";
    706: OLine4:= "O140_LK_TST6 _SEL5(Q706.3)    ";
    707: OLine4:= "O160_MC_LMP_ON(Q707.3)        ";
    708: OLine4:= "O160_BOT_MC_LMP_ON(Q708.3)    ";
    709: OLine4:= "O10B_ROB_MAN_AUTO_MODE(Q709.3)";
   1340: OLine4:= "O130_RH_ROTRY_180_DEG(Q1340.3)";
   1341: OLine4:= "O140_VERT_SUP1_CYL_FWD(Q1341.3)";
   1342: OLine4:= "O140_VERT_SUP2_CYL_FWD(Q1342.3)";
   1343: OLine4:= "O140_VERT_SUP3_CYL_FWD(Q1343.3)";
   1350: OLine4:= "O160_RH_COMP_PP_GRPR_CLSE_OPN(Q1350.3)";
   1351: OLine4:= "O160_LH_PALLET_LOCK_CYL_LOCK(Q1351.3)";
   1352: OLine4:= "OP160_MOVR_REM_CYL_FWD(Q1352.3)";
   1353: OLine4:= "O160_SPARE_Q1353_3(Q1353.3)";
    ELSE
      OLine4:= " ";	
    END_CASE
        Out_Visibility_4:=TRUE;
   
   CASE OP_Arr_OP160P[Output_Page_num] OF
	700:  Out_Lamp4:=O140_LK_TST1_SEL2_Q700_3;
	701:  Out_Lamp4:=O140_LK_TST2_SEL1_Q701_3;
	702:  Out_Lamp4:=O140_LK_TST3_STRT_Q702_3;
	703:  Out_Lamp4:=O140_LK_TST4_RST_Q703_3;
	704:  Out_Lamp4:=O140_LK_TST4_SEL7_Q704_3;
	705:  Out_Lamp4:=O140_LK_TST5_SEL6_Q705_3;
	706:  Out_Lamp4:=O140_LK_TST6_SEL5_Q706_3;
	707:  Out_Lamp4:=O160_MC_LMP_ON_Q707_3;
	708:  Out_Lamp4:=O160_BOT_MC_LMP_ON_Q708_3;
	709:  Out_Lamp4:=O10B_ROB_MAN_AUTO_MODE_Q709_3;
	1340: Out_Lamp4:=O130_RH_ROTRY_180_DEG_Q1340_3;
	1341: Out_Lamp4:=O140_VERT_SUP1_CYL_FWD_Q1341_3;
	1342: Out_Lamp4:=O140_VERT_SUP2_CYL_FWD_Q1342_3;
	1343: Out_Lamp4:=O140_VERT_SUP3_CYL_FWD_Q1343_3;
	1350: Out_Lamp4:=O160_RH_COMP_PP_GRPR_CLSE_OPN_Q1350_3;
	1351: Out_Lamp4:=O160_LH_PALLET_LOCK_CYL_LOCK_Q1351_3;
	1352: Out_Lamp4:= OP160_MOVR_REM_CYL_FWD_Q1352_3;
	1353: Out_Lamp4:=O160_SPARE_Q1353_3;
   ELSE
       Out_Visibility_4:=FALSE;
   END_CASE 
    
    CASE OP_Arr_OP160P[Output_Page_num] OF
    700: OLine5:= "O140_LK_TST1 _SEL3(Q700.4)     ";
    701: OLine5:= "O140_LK_TST2 _SEL2(Q701.4)     ";
    702: OLine5:= "O140_LK_TST3 _SEL1(Q702.4)     ";
    703: OLine5:= "O140_LK_TST4 _STRT(Q703.4)     ";
    704: OLine5:= "O140_LK_TST5_RST(Q704.4)       ";
    705: OLine5:= "O140_LK_TST5 _SEL7(Q705.4)     ";
    706: OLine5:= "O140_LK_TST6 _SEL6(Q706.4)     ";
    707: OLine5:= "O160_AUTOBAG_CNT_CMPLTD(Q707.4)";
    708: OLine5:= "O10A_DRUM_MTR_FWD(Q708.4)      ";
    709: OLine5:= "O120_ROB_MAN_AUTO_MODE(Q709.4) ";
   1340: OLine5:= "O130_LH_TOOL_CHO_UNLOCK(Q1340.4)";
   1341: OLine5:= "O140_TOOL1_CHO_UNLOCK(Q1341.4)";
   1342: OLine5:= "O140_TOOL2_CHO_UNLOCK(Q1342.4)";
   1343: OLine5:= "O140_TOOL3_CHO_UNLOCK(Q1343.4)";
   1350: OLine5:= "O160_SLIDE_CYL_REV(Q1350.4)";
   1351: OLine5:= "O160_RH_PALLET_LOCK_CYL_UNLOCK(Q1351.4)";
   1352: OLine5:= "O160_SPARE_Q1352_4(Q1352.4)";
   1353: OLine5:= "O160_SPARE_Q1353_4(Q1353.4)";
    ELSE
      OLine5:= " ";	
    END_CASE
       Out_Visibility_5:=TRUE;
	
    CASE OP_Arr_OP160P[Output_Page_num] OF
	700:  Out_Lamp5:=O140_LK_TST1_SEL3_Q700_4;
	701:  Out_Lamp5:=O140_LK_TST2_SEL2_Q701_4;
	702:  Out_Lamp5:=O140_LK_TST3_SEL1_Q702_4;
	703:  Out_Lamp5:=O140_LK_TST4_STRT_Q703_4;
	704:  Out_Lamp5:=O140_LK_TST5_RST_Q704_4;
	705:  Out_Lamp5:=O140_LK_TST5_SEL7_Q705_4;
	706:  Out_Lamp5:=O140_LK_TST6_SEL6_Q706_4;
	707:  Out_Lamp5:=O160_AUTOBAG_CNT_CMPLTD_Q707_4;
	708:  Out_Lamp5:=O10A_DRUM_MTR_FWD_Q708_4;
	709:  Out_Lamp5:=O120_ROB_MAN_AUTO_MODE_Q709_4;
	1340: Out_Lamp5:=O130_LH_TOOL_CHO_UNLOCK_Q1340_4;
	1341: Out_Lamp5:=O140_TOOL1_CHO_UNLOCK_Q1341_4;
	1342: Out_Lamp5:=O140_TOOL2_CHO_UNLOCK_Q1342_4;
	1343: Out_Lamp5:=O140_TOOL3_CHO_UNLOCK_Q1343_4;
	1350: Out_Lamp5:=O160_SLIDE_CYL_REV_Q1350_4;
	1351: Out_Lamp5:=O160_RH_PALLET_LOCK_CYL_UNLOCK_Q1351_4;
	1352: Out_Lamp5:=O160_SPARE_Q1352_4;
	1353: Out_Lamp5:=O160_SPARE_Q1353_4;
   ELSE
       Out_Visibility_5:=FALSE;
   END_CASE 
    
    CASE OP_Arr_OP160P[Output_Page_num] OF
    700: OLine6:= "O140_LK_TST1 _SEL4(Q700.5)        ";
    701: OLine6:= "O140_LK_TST2 _SEL3(Q701.5)        ";
    702: OLine6:= "O140_LK_TST3 _SEL2(Q702.5)        ";
    703: OLine6:= "O140_LK_TST4 _SEL1(Q703.5)        ";
    704: OLine6:= "O140_LK_TST5 _STRT(Q704.5)        ";
    705: OLine6:= "O140_LK_TST6 _RST(Q705.5)         ";
    706: OLine6:= "O140_LK_TST6 _SEL7(Q706.5)        ";
    707: OLine6:= "O160_SAMPLE_PART_DOR_OPN(Q707.5) ";
    708: OLine6:= "O10A_DRUM_RST(Q708.5)             ";
    709: OLine6:= "O160_SPARE_Q709_5(Q709.5)         ";
   1340: OLine6:= "O130_LH_TOOL_CHO_LOCK(Q1340.5)";
   1341: OLine6:= "O140_TOOL1_CHO_LOCK(Q1341.5)";
   1342: OLine6:= "O140_TOOL2_CHO_LOCK(Q1342.5)";
   1343: OLine6:= "O140_TOOL3_CHO_LOCK(Q1343.5)";
   1350: OLine6:= "O160_SLIDE_CYL_FWD(Q1350.5)";
   1351: OLine6:= "O160_RH_PALLET_LOCK_CYL_LOCK(Q1351.5)";
   1352: OLine6:= "O160_SPARE_Q1352_5(Q1352.5)";
   1353: OLine6:= "O160_SPARE_Q1353_5(Q1353.5)";
    ELSE
      OLine6:= " ";	
    END_CASE
       Out_Visibility_6:=TRUE;
	
    CASE OP_Arr_OP160P[Output_Page_num] OF
	700:  Out_Lamp6:=O140_LK_TST1_SEL4_Q700_5;
	701:  Out_Lamp6:=O140_LK_TST2_SEL3_Q701_5;
	702:  Out_Lamp6:=O140_LK_TST3_SEL2_Q702_5;
	703:  Out_Lamp6:=O140_LK_TST4_SEL1_Q703_5;
	704:  Out_Lamp6:=O140_LK_TST5_STRT_Q704_5;
	705:  Out_Lamp6:=O140_LK_TST6_RST_Q705_5;
	706:  Out_Lamp6:=O140_LK_TST6_SEL7_Q706_5;
	707:  Out_Lamp6:=O160_SAMPLE_PART_DOOR_OPN_Q707_5;
	708:  Out_Lamp6:=O10A_DRUM_RST_Q708_5;
	709:  Out_Lamp6:=O160_SPARE_Q709_5;
	1340: Out_Lamp6:=O130_LH_TOOL_CHO_LOCK_Q1340_5;
	1341: Out_Lamp6:=O140_TOOL1_CHO_LOCK_Q1341_5;
	1342: Out_Lamp6:=O140_TOOL2_CHO_LOCK_Q1342_5;
	1343: Out_Lamp6:=O140_TOOL3_CHO_LOCK_Q1343_5;
	1350: Out_Lamp6:=O160_SLIDE_CYL_FWD_Q1350_5;
	1351: Out_Lamp6:=O160_RH_PALLET_LOCK_CYL_LOCK_Q1351_5;
	1352: Out_Lamp6:=O160_SPARE_Q1352_5;
	1353: Out_Lamp6:=O160_SPARE_Q1353_5;
   ELSE           
       Out_Visibility_6:=FALSE;
   END_CASE 
       
    CASE OP_Arr_OP160P[Output_Page_num] OF
    700: OLine7:= "O140_LK_TST1 _SEL5(Q700.6)    ";
    701: OLine7:= "O140_LK_TST2 _SEL4(Q701.6)    ";
    702: OLine7:= "O140_LK_TST3 _SEL3(Q702.6)    ";
    703: OLine7:= "O140_LK_TST4 _SEL2(Q703.6)    ";
    704: OLine7:= "O140_LK_TST5 _SEL1(Q704.6)    ";
    705: OLine7:= "O140_LK_TST6 _STRT(Q705.6)    ";
    706: OLine7:= "O150_VISN_LGHT_ON(Q706.6)     ";
    707: OLine7:= "O160_REJ_BIN_DOR_OPN(Q707.6) ";
    708: OLine7:= "O10A_DRUM_EXT_SPEED(Q708.6)   ";
    709: OLine7:= "O160_SPARE_Q709_6(Q709.6)     ";
   1340: OLine7:= "O130_RH_TOOL_CHO_UNLOCK(Q1340.6)";
   1341: OLine7:= "O140_WIPE1_CYL_REV(Q1341.6)";
   1342: OLine7:= "O140_WIPE2_CYL_REV(Q1342.6)";
   1343: OLine7:= "O140_WIPE3_CYL_REV(Q1343.6)";
   1350: OLine7:= "O160_SPARE_Q1350_6(Q1350.6)";
   1351: OLine7:= "O160_SPARE_Q1351_6(Q1351.6)";
   1352: OLine7:= "O160_SPARE_Q1352_6(Q1352.6)";
   1353: OLine7:= "O160_SPARE_Q1353_6(Q1353.6)";
    ELSE
      OLine7:= " ";	
    END_CASE
       Out_Visibility_7:=TRUE;
	
   CASE OP_Arr_OP160P[Output_Page_num] OF
	700:  Out_Lamp7:=O140_LK_TST1_SEL5_Q700_6;
	701:  Out_Lamp7:=O140_LK_TST2_SEL4_Q701_6;
	702:  Out_Lamp7:=O140_LK_TST3_SEL3_Q702_6;
	703:  Out_Lamp7:=O140_LK_TST4_SEL2_Q703_6;
	704:  Out_Lamp7:=O140_LK_TST5_SEL1_Q704_6;
	705:  Out_Lamp7:=O140_LK_TST6_STRT_Q705_6;
	706:  Out_Lamp7:=O150_VISN_LGHT_ON_Q706_6;
	707:  Out_Lamp7:=O160_REJ_BIN_DOOR_OPN_Q707_6;
	708:  Out_Lamp7:=O10A_DRUM_EXT_SPEED_Q708_6;
	709:  Out_Lamp7:=O160_SPARE_Q709_6;
	1340: Out_Lamp7:=O130_RH_TOOL_CHO_UNLOCK_Q1340_6;
	1341: Out_Lamp7:=O140_WIPE1_CYL_REV_Q1341_6;
	1342: Out_Lamp7:=O140_WIPE2_CYL_REV_Q1342_6;
	1343: Out_Lamp7:=O140_WIPE3_CYL_REV_Q1343_6;
	1350: Out_Lamp7:=O160_SPARE_Q1350_6;
	1351: Out_Lamp7:=O160_SPARE_Q1351_6;
	1352: Out_Lamp7:=O160_SPARE_Q1352_6;
	1353: Out_Lamp7:=O160_SPARE_Q1353_6;
   ELSE
       Out_Visibility_7:=FALSE;
   END_CASE 
    
    CASE OP_Arr_OP160P[Output_Page_num] OF
    700: OLine8:= "O140_LK_TST1_SEL6(Q700.7)";
    701: OLine8:= "O140_LK_TST2_SEL5(Q701.7)";
    702: OLine8:= "O140_LK_TST3_SEL4(Q702.7)";
    703: OLine8:= "O140_LK_TST4_SEL3(Q703.7)";
    704: OLine8:= "O140_LK_TST5_SEL2(Q704.7)";
    705: OLine8:= "O140_LK_TST6_SEL1(Q705.7)";
    706: OLine8:= "O150_BARLIGHT_OP1(Q706.7) ";
    707: OLine8:= "O160_SPARE(Q707.7)        ";
    708: OLine8:= "O160_SPARE_Q708_7(Q708.7) ";
    709: OLine8:= "O160_SPARE_Q709_7(Q709.7) ";
   1340: OLine8:= "O130_RH_TOOL_CHO_LOCK(Q1340.7)";
   1341: OLine8:= "O140_WIPE1_CYL_FWD(Q1341.7)";
   1342: OLine8:= "O140_WIPE2_CYL_FWD(Q1342.7)";
   1343: OLine8:= "O140_WIPE3_CYL_FWD(Q1343.7)";
   1350: OLine8:= "O160_SPARE_Q1350_7(Q1350.7)";
   1351: OLine8:= "O160_SPARE_Q1351_7(Q1351.7)";
   1352: OLine8:= "O160_SPARE_Q1352_7(Q1352.7)";
   1353: OLine8:= "O160_SPARE_Q1353_7(Q1353.7)";
    ELSE
      OLine8:= " ";	
    END_CASE	
       Out_Visibility_8:=TRUE;
   
   CASE OP_Arr_OP160P[Output_Page_num] OF
	700:  Out_Lamp8:=O140_LK_TST1_SEL6_Q700_7;
	701:  Out_Lamp8:=O140_LK_TST2_SEL5_Q701_7;
	702:  Out_Lamp8:=O140_LK_TST3_SEL4_Q702_7;
	703:  Out_Lamp8:=O140_LK_TST4_SEL3_Q703_7;
	704:  Out_Lamp8:=O140_LK_TST5_SEL2_Q704_7;
	705:  Out_Lamp8:=O140_LK_TST6_SEL1_Q705_7;
	706:  Out_Lamp8:=O150_BARLIGHT_OP1_Q706_7;
	707:  Out_Lamp8:=O160_SPARE_Q707_7;
	708:  Out_Lamp8:=O160_SPARE_Q708_7;
	709:  Out_Lamp8:=O160_SPARE_Q709_7;
	1340: Out_Lamp8:=O130_RH_TOOL_CHO_LOCK_Q1340_7;
	1341: Out_Lamp8:=O140_WIPE1_CYL_FWD_Q1341_7;
	1342: Out_Lamp8:=O140_WIPE2_CYL_FWD_Q1342_7;
	1343: Out_Lamp8:=O140_WIPE3_CYL_FWD_Q1343_7;
	1350: Out_Lamp8:=O160_SPARE_Q1350_7;
	1351: Out_Lamp8:=O160_SPARE_Q1351_7;
	1352: Out_Lamp8:=O160_SPARE_Q1352_7;
	1353: Out_Lamp8:=O160_SPARE_Q1353_7;
   ELSE
       Out_Visibility_8:=FALSE;	
   END_CASE 
  
 4: CASE IP_Arr_OP10A[Input_Page_num] OF
      100:Line1:="I10A_HPR_UNIT_ALRM(I100.0)    ";
      101:Line1:="I10A_HPR_DOOR_SELCTN(I101.0)  ";
      102:Line1:="I10A_LNR_TRK1_CHO_MOD1(I102.0)";
      103:Line1:="I10A_SPARE_I103_0(I103.0)     ";
      ELSE
      	Line1:= " ";
      END_CASE
      
      CASE IP_Arr_OP10A[Input_Page_num] OF
      100:Line2:="I10A_SPARE_I100.1(I100.1)      ";
      101:Line2:="I10A_SPARE_I101.1(I101.1)      ";
      102:Line2:="I10A_LNR_TRK1_CHO_MOD2(I102.1) ";
      103:Line2:="I10A_SPARE_I103_1(I103.1)      ";
      ELSE
      	Line2 := " ";
      END_CASE
      
      CASE IP_Arr_OP10A[Input_Page_num] OF
      100:Line3:="I10A_HPR_LOW_LVL_SEN(I100.2)   ";
      101:Line3:="I10A_BDY_BOWL_LOW_LVL(I101.2)  ";
      102:Line3:="I10A_LNR_TRK2_CHO_MOD1(I102.2) ";
      103:Line3:="I10A_SPARE_I103_2(I103.2)      ";
      ELSE
      	Line3 := " ";
      END_CASE
      
      CASE IP_Arr_OP10A[Input_Page_num] OF
      100:Line4:="I10A_HPR_SOL_DOOR_SW_FB(I100.3)";
      101:Line4:="I10A_BDY_BWL_RUN(I101.3)       ";
      102:Line4:="I10A_LNR_TRK2_CHO_MOD2(I102.3) ";
      103:Line4:="I10A_SPARE_I103_3(I103.3)      ";
      ELSE
      	Line4 := " ";
      END_CASE
      
      CASE IP_Arr_OP10A[Input_Page_num] OF
      100:Line5:="I10A_HPR_OFF_ON(I100.4)";
      101:Line5:="I10A_BDY_LNR1_RUN(I101.4)";
      102:Line5:="I10A_SPARE_I102_4(I102.4)";
      103:Line5:="I10A_SPARE_I103_4(I103.4)";
      ELSE
      	Line5:= " ";
      END_CASE
      
      CASE IP_Arr_OP10A[Input_Page_num] OF
      100:Line6:="I10A_BDY_BOWL_OFF_ON(I100.5)  ";
      101:Line6:="I10A_BDY_LNR2_RUN(I101.5)     ";
      102:Line6:="I10A_SPARE_I102_5(I102.5)";
      103:Line6:="I10A_SPARE_I103_5(I103.5)     ";
      ELSE
      	Line6 := " ";
      END_CASE
      
      CASE IP_Arr_OP10A[Input_Page_num] OF
      100:Line7:="I10A_BDY_LNR1_OFF_ON(I100.6)     ";
      101:Line7:="I10A_BDY_LNR_FEED1_OVRFLW(I101.6)";
      102:Line7:="I10A_LH_BDY_CONT_FB(I102.6)      ";
      103:Line7:="I10A_SPARE_I103_6(I103.6)        ";
      ELSE
      	Line7 := " ";
      END_CASE
      
      CASE IP_Arr_OP10A[Input_Page_num] OF
      100:Line8:="I10A_BDY_LNR2_OFF_ON(I100.7)     ";
      101:Line8:="I10A_BDY_LNR_FEED2_OVRFLW(I101.7)";
      102:Line8:="I10A_RH_BDY_CONT_FB(I102.7)      ";
      103:Line8:="I10A_SPARE_I103_7(I103.7)        ";
      ELSE
      	Line8 := " ";
      END_CASE
	 	Visibility_1:=TRUE;
   
   CASE IP_Arr_OP10A[Input_Page_num] OF
	100: Lamp1:=I10A_HPR_UNIT_ALRM_I100_0 ;
	101: Lamp1:=I10A_HPR_DOOR_SELCTN_I101_0 ;
	102: Lamp1:=I10A_LNR_TRK1_CHO_MOD1_I102_0 ;
	103: Lamp1:=I10A_SPARE_I103_0;
   ELSE
       Visibility_1:=FALSE;	
   END_CASE
   
   Visibility_2:=TRUE;
   
   CASE IP_Arr_OP10A[Input_Page_num] OF
	100: Lamp2:=I10A_SPARE_I100_1 ;
	101: Lamp2:=I10A_SPARE_I101_1;
	102: Lamp2:=I10A_LNR_TRK1_CHO_MOD2_I102_1 ;
	103: Lamp2:=I10A_SPARE_I103_1;
   ELSE
       Visibility_2:=FALSE;	
   END_CASE
   
   
    Visibility_3:=TRUE;
   
   CASE IP_Arr_OP10A[Input_Page_num] OF
	100: Lamp3:=I10A_HPR_LOW_LVL_SEN_I100_2 ;
	101: Lamp3:=I10A_BDY_BOWL_LOW_LVL_I101_2 ;
	102: Lamp3:=I10A_LNR_TRK2_CHO_MOD1_I102_2 ;
	103: Lamp3:=I10A_SPARE_I103_2;
   ELSE
       Visibility_3:=FALSE;	
   END_CASE
   
   
    Visibility_4:=TRUE;
   
   CASE IP_Arr_OP10A[Input_Page_num] OF
	100: Lamp4:=I10A_HPR_SOL_DOOR_SW_FB_I100_3 ;
	101: Lamp4:=I10A_BDY_BWL_RUN_I101_3 ;
	102: Lamp4:=I10A_LNR_TRK2_CHO_MOD2_I102_3 ;
	103: Lamp4:=I10A_SPARE_I103_3;
   ELSE
       Visibility_4:=FALSE;	
   END_CASE
   
   
    
    Visibility_5:=TRUE;
   
   CASE IP_Arr_OP10A[Input_Page_num] OF
	100: Lamp5:=I10A_HPR_OFF_ON_I100_4 ;
	101: Lamp5:=I10A_BDY_LNR1_RUN_I101_4 ;
	102: Lamp5:=I10A_SPARE_I102_4 ;
	103: Lamp5:=I10A_SPARE_I103_4;
   ELSE
       Visibility_5:=FALSE;	
   END_CASE
   
    
    Visibility_6:=TRUE;
   
   CASE IP_Arr_OP10A[Input_Page_num] OF
	100: Lamp6:=I10A_BDY_BOWL_OFF_ON_I100_5 ;
	101: Lamp6:=I10A_BDY_LNR2_RUN_I101_5 ;
	102: Lamp6:=I10A_SPARE_I102_5 ;
	103: Lamp6:=I10A_SPARE_I103_5;
   ELSE
       Visibility_6:=FALSE;	
   END_CASE
   
   
      
    Visibility_7:=TRUE;
   
   CASE IP_Arr_OP10A[Input_Page_num] OF
	100: Lamp7:=I10A_BDY_LNR1_OFF_ON_I100_6 ;
	101: Lamp7:=I10A_BDY_LNR_FEED1_OVRFLW_I101_6 ;
	102: Lamp7:=I10A_LH_BDY_CONT_FB_I102_6;
	103: Lamp7:=I10A_SPARE_I103_6;
   ELSE
       Visibility_7:=FALSE;	
   END_CASE


 	Visibility_8:=TRUE;
   
   CASE IP_Arr_OP10A[Input_Page_num] OF
	100: Lamp8:=I10A_BDY_LNR2_OFF_ON_I100_7 ;
	101: Lamp8:=I10A_BDY_LNR_FEED2_OVRFLW_I101_7 ;
	102: Lamp8:=I10A_RH_BDY_CONT_FB_I102_7 ;
	103: Lamp8:=I10A_SPARE_I103_7;
   ELSE
       Visibility_8:=FALSE;	
   END_CASE

	
	 CASE OP_Arr_OP10A[Output_Page_num] OF
     100:OLine1:="O10A_HPR_MTR_FWD(Q100.0)  ";
     101:OLine1:="O10A_BDY_BOWL_ON(Q101.0)  ";
     102:OLine1:="O10A_SPARE_Q102_0(Q102.0) ";
     103:OLine1:="O10A_SPARE_Q103_0(Q103.0) ";
     ELSE
     	OLine1:= " ";
     END_CASE
     
     CASE OP_Arr_OP10A[Output_Page_num] OF
     100:OLine2:="O10A_HPR_RST(Q100.1)         ";
     101:OLine2:="O10A_BDY_LNR_FEED1_ON(Q101.1)";
     102:OLine2:="O10A_SPARE_Q102_1(Q102.1)    ";
     103:OLine2:="O10A_SPARE_Q103_1(Q103.1)    ";
     ELSE
     	OLine2:= " ";
     END_CASE
     
     CASE OP_Arr_OP10A[Output_Page_num] OF
     100:OLine3:="O10A_EXT_SPEED(Q100.2)       ";
     101:OLine3:="O10A_BDY_LNR_FEED2_ON(Q101.2)";
     102:OLine3:="O10A_SPARE_Q102_2(Q102.2)    ";
     103:OLine3:="O10A_SPARE_Q103_2(Q103.2)    ";
     ELSE
     	OLine3:= " ";
     END_CASE
     
     CASE OP_Arr_OP10A[Output_Page_num] OF
     100:OLine4:="O10A_SPARE_Q100.3(Q100.3)      ";
     101:OLine4:="O10A_BDY_LNR1_AIR_PURGE(Q101.3)";
     102:OLine4:="O10A_SPARE_Q102_3(Q102.3)      ";
     103:OLine4:="O10A_SPARE_Q103_3(Q103.3)      ";
     ELSE
     	OLine4:= " ";
     END_CASE
     
     CASE OP_Arr_OP10A[Output_Page_num] OF
     100:OLine5:="O10A_HPR_DOOR_SELCTN_IND(Q100.4)";
   //101:OLine5:="O10A_BDY_LNR2_AIRPURGE(Q101.4)";
     102:OLine5:="O10A_SPARE_Q102_4(Q102.4)";
     103:OLine5:="O10A_SPARE_Q103_4(Q103.4)";
     ELSE
     	OLine5:= " ";
     END_CASE
     
     CASE OP_Arr_OP10A[Output_Page_num] OF
     100:OLine6:="O10A_HPR_TWR_LMP_RED(Q100.5)";
     101:OLine6:="O10A_HPR_DOOR_OPN(Q101.5)   ";
     102:OLine6:="O10A_SPARE_Q102_5(Q102.5)   ";
     103:OLine6:="O10A_SPARE_Q103_5(Q103.5)   ";
     ELSE
     	OLine6:= " ";
     END_CASE
     
     CASE OP_Arr_OP10A[Output_Page_num] OF
     100:OLine7:="O10A_HPR_TWR_LMP_GREEN(Q100.6)";
     101:OLine7:="O10A_SPARE_Q101_6(Q101.6)     ";
     102:OLine7:="O10A_SPARE_Q102_6(Q102.6)     ";
     103:OLine7:="O10A_SPARE_Q103_6(Q103.6)     ";
     ELSE
     	OLine7:= " ";
     END_CASE
     
     CASE OP_Arr_OP10A[Output_Page_num] OF
     100:OLine8:="O10A_SPARE_Q100_7(Q100.7)";
     101:OLine8:="O10A_SPARE_Q101_7(Q101.7)";
     102:OLine8:="O10A_SPARE_Q102_7(Q102.7)";
     103:OLine8:="O10A_SPARE_Q103_7(Q103.7)";
     ELSE
     	OLine8:= " ";
     END_CASE
	  Out_Visibility_1:=TRUE;

    CASE OP_Arr_OP10A[Output_Page_num] OF
	100:  Out_Lamp1:=O10A_HPR_MTR_FWD_Q100_0;
	101:  Out_Lamp1:=O10A_BDY_BOWL_ON_Q101_0;
	102:  Out_Lamp1:=O10A_SPARE_Q102_0;
	103:  Out_Lamp1:=O10A_SPARE_Q103_0;
   ELSE
       Out_Visibility_1:=FALSE;	
   END_CASE
   
    Out_Visibility_2:=TRUE;
   
   CASE OP_Arr_OP10A[Output_Page_num] OF
	100:  Out_Lamp2:=O10A_HPR_RST_Q100_1;
	101:  Out_Lamp2:=O10A_BDY_LNR_FEED1_ON_Q101_1;
	102:  Out_Lamp2:=O10A_SPARE_Q102_1;
	103:  Out_Lamp2:=O10A_SPARE_Q103_1;
   ELSE
       Out_Visibility_2:=FALSE;	
   END_CASE 
   
    Out_Visibility_3:=TRUE;
	
   CASE OP_Arr_OP10A[Output_Page_num] OF
	100:  Out_Lamp3:=O10A_EXT_SPEED_Q100_2; 
	101:  Out_Lamp3:=O10A_BDY_LNR_FEED2_ON_Q101_2; 
	102:  Out_Lamp3:=O10A_SPARE_Q102_2; 
	103:  Out_Lamp3:=O10A_SPARE_Q103_2; 
   ELSE
       Out_Visibility_3:=FALSE;
   END_CASE 
   
    Out_Visibility_4:=TRUE;
   
   CASE OP_Arr_OP10A[Output_Page_num] OF
	100:  Out_Lamp4:=O10A_SPARE_Q100_3; 
	101:  Out_Lamp4:=O10A_BDY_LNR1_AIR_PURGE_Q101_3; 
	102:  Out_Lamp4:=O10A_SPARE_Q102_3; 
	103:  Out_Lamp4:=O10A_SPARE_Q103_3;  
   ELSE
       Out_Visibility_4:=FALSE;
   END_CASE 
   
    Out_Visibility_5:=TRUE;
	
    CASE OP_Arr_OP10A[Output_Page_num] OF
	100:  Out_Lamp5:=O10A_HPR_DOOR_SELCTN_IND_Q100_4; 
	//101:  Out_Lamp5:=O10A_BDY_LNR2_AIR_PURGE_Q101_4; 
	102:  Out_Lamp5:=O10A_SPARE_Q102_4; 
	103:  Out_Lamp5:=O10A_SPARE_Q103_4; 	 
   ELSE
       Out_Visibility_5:=FALSE;
   END_CASE 
   
    Out_Visibility_6:=TRUE;
	
   CASE OP_Arr_OP10A[Output_Page_num] OF
	100:  Out_Lamp6:=O10A_HPR_TWR_LMP_RED_Q100_5; 
	101:  Out_Lamp6:=O10A_HPR_DOOR_OPN_Q101_5; 
	102:  Out_Lamp6:=O10A_SPARE_Q102_5; 
	103:  Out_Lamp6:=O10A_SPARE_Q103_5; 
   ELSE           
       Out_Visibility_6:=FALSE;
   END_CASE 
    
	Out_Visibility_7:=TRUE;
	
   CASE OP_Arr_OP10A[Output_Page_num] OF
	100:  Out_Lamp7:=O10A_HPR_TWR_LMP_GREEN_Q100_6; 
	101:  Out_Lamp7:=O10A_SPARE_Q101_6; 
	102:  Out_Lamp7:=O10A_SPARE_Q102_6; 
	103:  Out_Lamp7:=O10A_SPARE_Q103_6;  
   ELSE 
       Out_Visibility_7:=FALSE;
   END_CASE 
   
    Out_Visibility_8:=TRUE;
   
   CASE OP_Arr_OP10A[Output_Page_num] OF
	100:  Out_Lamp8:=O10A_SPARE_Q100_7;  
	101:  Out_Lamp8:=O10A_SPARE_Q101_7;  
	102:  Out_Lamp8:=O10A_SPARE_Q102_7;  
	103:  Out_Lamp8:=O10A_SPARE_Q103_7;   
   ELSE
       Out_Visibility_8:=FALSE;	
   END_CASE
	 
 5: CASE IP_Arr_OP10B[Input_Page_num] OF
    200: Line1:= "I10B_HPR_UNIT_ALRM(I200.0)     ";
    201: Line1:= "I10B_HPR_DOOR_SELCTN(I201.0)   ";
    202: Line1:= "I10B_LNR_TRK1_CHO_MOD1(I202.0) ";
    203: Line1:= "I10B_SPARE_I203_0(I203.0)      ";
    ELSE
    	Line1 := " ";
    END_CASE
    
    CASE IP_Arr_OP10B[Input_Page_num] OF
    200: Line2:= "I10B_SPARE_I200_1(I200.1)     ";
    201: Line2:= "I10B_SPARE_I201_1(I201.1)     ";
    202: Line2:= "I10B_LNR_TRK1_CHO_MOD2(I202.1)";
    203: Line2:= "I10B_SPARE_I203_1(I203.1)     ";
    ELSE
    	Line2 := " ";
    END_CASE
    
    CASE IP_Arr_OP10B[Input_Page_num] OF
    200: Line3:= "I10B_HPR_LOW_LVL_SEN(I200.2)   ";
    201: Line3:= "I10B_BDY_BOWL_LOW_LVL(I201.2)  ";
    202: Line3:= "I10B_LNR_TRK2_CHO_MOD1(I202.2) ";
    203: Line3:= "I10B_SPARE_I203_2(I203.2)      ";
    ELSE
    	Line3 := " ";
    END_CASE
    
    CASE IP_Arr_OP10B[Input_Page_num] OF
    200: Line4:= "I10B_HPR_SOL_DOOR_SW_FB(I200.3)";
    201: Line4:= "I10B_BDY_BWL_RUN(I201.3)       ";
    202: Line4:= "I10B_LNR_TRK2_CHO_MOD2(I202.3) ";
    203: Line4:= "I10B_SPARE_I203_3(I203.3)      ";
    ELSE
    	Line4 := " ";
    END_CASE
    
    CASE IP_Arr_OP10B[Input_Page_num] OF
    200: Line5:= "I10B_HPR_OFF_ON(I200.4)       ";
    201: Line5:= "I10B_BDY_LNR1_RUN(I201.4)     ";
    202: Line5:= "I10B_SPARE_I202_4(I202.4)";
    203: Line5:= "I10B_SPARE_I203_4(I203.4)     ";
    ELSE
    	Line5 := " ";
    END_CASE
    
    CASE IP_Arr_OP10B[Input_Page_num] OF
    200: Line6:= "I10B_BDY_BOWL_OFF_ON(I200.5)   ";
    201: Line6:= "I10B_BDY_LNR2_RUN(I201.5)      ";
    202: Line6:= "I10B_SPARE_I202_5(I202.5) ";
    203: Line6:= "I10B_SPARE_I203_5(I203.5)      ";
    ELSE
    	Line6 := " ";
    END_CASE
    
    CASE IP_Arr_OP10B[Input_Page_num] OF
    200: Line7:= "I10B_BDY_LNR1_OFF_ON(I200.6)      ";
    201: Line7:= "I10B_BDY_LNR_FEED1_OVRFLW(I201.6) ";
    202: Line7:= "I10B_SPARE_I202_6(I202.6)         ";
    203: Line7:= "I10B_SPARE_I203_6(I203.6)         ";
    ELSE
    	Line7 := " ";
    END_CASE
    
    CASE IP_Arr_OP10B[Input_Page_num] OF
    200: Line8:= "I10B_BDY_LNR2_OFF_ON(I200.7)     ";
    201: Line8:= "I10B_BDY_LNR_FEED2_OVRFLW(I201.7)";
    202: Line8:= "I10B_SPARE_I202_7(I202.7)        ";
    203: Line8:= "I10B_SPARE_I203_7(I203.7)        ";
    ELSE
    	Line8 := " ";
    END_CASE
	  Visibility_1:=TRUE;
   
   CASE IP_Arr_OP10B[Input_Page_num] OF
	200: Lamp1:=I10B_HPR_UNIT_ALRM_I200_0 ;
	201: Lamp1:=I10B_HPR_DOOR_SELCTN_I201_0 ;
	202: Lamp1:=I10B_LNR_TRK1_CHO_MOD1_I202_0 ;
	203: Lamp1:=I10B_SPARE_I203_0;
   ELSE
       Visibility_1:=FALSE;	
   END_CASE
   
   
   Visibility_2:=TRUE;
   
   CASE IP_Arr_OP10B[Input_Page_num] OF
	200: Lamp2:=I10B_SPARE_I200_1 ;
	201: Lamp2:=I10B_SPARE_I201_1 ;
	202: Lamp2:=I10B_LNR_TRK1_CHO_MOD2_I202_1 ;
	203: Lamp2:=I10B_SPARE_I203_1;
   ELSE
       Visibility_2:=FALSE;	
   END_CASE
   
   
    Visibility_3:=TRUE;
   
   CASE IP_Arr_OP10B[Input_Page_num] OF
	200: Lamp3:=I10B_HPR_LOW_LVL_SEN_I200_2 ;
	201: Lamp3:=I10B_BDY_BOWL_LOW_LVL_I201_2 ; 
	202: Lamp3:=I10B_LNR_TRK2_CHO_MOD1_I202_2 ;
	203: Lamp3:=I10B_SPARE_I203_2 ;
   ELSE
       Visibility_3:=FALSE;	
   END_CASE
   
   
    Visibility_4:=TRUE;
   
   CASE IP_Arr_OP10B[Input_Page_num] OF
	200: Lamp4:=I10B_HPR_SOL_DOOR_SW_FB_I200_3 ;
	201: Lamp4:=I10B_BDY_BWL_RUN_I201_3 ; 
	202: Lamp4:=I10B_LNR_TRK2_CHO_MOD2_I202_3 ;
	203: Lamp4:=I10B_SPARE_I203_3 ;
   ELSE
       Visibility_4:=FALSE;	
   END_CASE
   
   
    Visibility_5:=TRUE;
   
   CASE IP_Arr_OP10B[Input_Page_num] OF
	200: Lamp5:=I10B_HPR_OFF_ON_I200_4 ;
	201: Lamp5:=I10B_BDY_LNR1_RUN_I201_4 ;
	202: Lamp5:=I10B_SPARE_I202_4 ;
	203: Lamp5:=I10B_SPARE_I203_4;
   ELSE
       Visibility_5:=FALSE;	
   END_CASE
   
    
    Visibility_6:=TRUE;
   
   CASE IP_Arr_OP10B[Input_Page_num] OF
	200: Lamp6:=I10B_BDY_BOWL_OFF_ON_I200_5 ;
	201: Lamp6:=I10B_BDY_LNR2_RUN_I201_5 ;
	202: Lamp6:=I10B_SPARE_I202_5 ;
	203: Lamp6:=I10B_SPARE_I203_5 ;
   ELSE
       Visibility_6:=FALSE;	
   END_CASE
   
      
    Visibility_7:=TRUE;
   
   CASE IP_Arr_OP10B[Input_Page_num] OF
	200: Lamp7:=I10B_BDY_LNR1_OFF_ON_I200_6 ;
	201: Lamp7:=I10B_BDY_LNR_FEED1_OVRFLW_I201_6 ;
	202: Lamp7:=I10B_SPARE_I202_6 ;
	203: Lamp7:=I10B_SPARE_I203_6;
   ELSE
       Visibility_7:=FALSE;	
   END_CASE


    Visibility_8:=TRUE;
   
   CASE IP_Arr_OP10B[Input_Page_num] OF
	200: Lamp8:=I10B_BDY_LNR2_OFF_ON_I200_7 ;
	201: Lamp8:=I10B_BDY_LNR_FEED2_OVRFLW_I201_7 ;
	202: Lamp8:=I10B_SPARE_I202_7 ;
	203: Lamp8:=I10B_SPARE_I203_7;
   ELSE
       Visibility_8:=FALSE;	
   END_CASE


  CASE OP_Arr_OP10B_JB[Output_Page_num] OF	
  200: OLine1:= " O10B_HPR_MTR_FWD(Q200.0) ";
  201: OLine1:= " O10B_BDY_BOWL_ON(Q201.0) ";
  202: OLine1:= " O10B_SPARE_Q202_0(Q202.0)";
  203: OLine1:= " O10B_SPARE_Q203_0(Q203.0)";
  ELSE
      OLine1 := " ";
  END_CASE
  
  CASE OP_Arr_OP10B_JB[Output_Page_num] OF
  200: OLine2:= "O10B_HPR_RST(Q200.1)         ";
  201: OLine2:= "O10B_BDY_LNR_FEED1_ON(Q201.1)";
  202: OLine2:= "O10B_SPARE_Q202_1(Q202.1)    ";
  203: OLine2:= "O10B_SPARE_Q203_1(Q203.1)    ";
  ELSE
    OLine2 := " ";
  END_CASE
  
  CASE OP_Arr_OP10B_JB[Output_Page_num] OF
  200: OLine3:= "O10B_EXT_SPEED(Q200.2)       ";
  201: OLine3:= "O10B_BDY_LNR_FEED2_ON(Q201.2)";
  202: OLine3:= "O10B_SPARE_Q202_2(Q202.2)    ";
  203: OLine3:= "O10B_SPARE_Q2032_(Q203.2)    ";
  ELSE
    OLine3 := " ";
  END_CASE
  
  CASE OP_Arr_OP10B_JB[Output_Page_num] OF
  200: OLine4:= "O10B_SPARE_Q200.3(Q200.3)      ";
  201: OLine4:= "O10B_BDY_LNR1_AIR_PURGE(Q201.3)";
  202: OLine4:= "O10B_SPARE_Q202_3(Q202.3)      ";
  203: OLine4:= "O10B_SPARE_Q203_3(Q203.3)      ";
  ELSE
    OLine4 := " ";
  END_CASE
  
  CASE OP_Arr_OP10B_JB[Output_Page_num] OF
  200: OLine5:= "O10B_HPR_DOOR_SELCTN_IND(Q200.4)";
  //201: OLine5:= "O10B_BDY_LNR2_AIR_PURGE(Q201.4) ";
  202: OLine5:= "O10B_SPARE_Q202_4(Q202.4)       ";
  203: OLine5:= "O10B_SPARE_Q203_4(Q203.4)       ";
  ELSE
     OLine5 := " ";
  END_CASE
  
  CASE OP_Arr_OP10B_JB[Output_Page_num] OF
  200: OLine6:= "O10B_HPR_TWR_LMP_RED(Q200.5)";
  201: OLine6:= "O10B_HPR_DOOR_OPN(Q201.5)   ";
  202: OLine6:= "O10B_SPARE_Q202_5(Q202.5)   ";
  203: OLine6:= "O10B_SPARE_Q203_5(Q203.5)   ";
  ELSE
     OLine6 := " ";
  END_CASE
  
  CASE OP_Arr_OP10B_JB[Output_Page_num] OF
  200: OLine7:= "O10B_HPR_TWR_LMP_GREEN(Q200.6)";
  201: OLine7:= "O10B_SPARE_Q201_6(Q201.6)     ";
  202: OLine7:= "O10B_SPARE_Q202_6(Q202.6)     ";
  203: OLine7:= "O10B_SPARE_Q203_6(Q203.6)     ";
  ELSE
      OLine7 := " ";
  END_CASE
  
  CASE OP_Arr_OP10B_JB[Output_Page_num] OF	 
  200: OLine8:= "O10B_SPARE_Q200_7(Q200.7)";
  201: OLine8:= "O10B_SPARE_Q201_7(Q201.7)";
  202: OLine8:= "O10B_SPARE_Q202_7(Q202.7)";
  203: OLine8:= "O10B_SPARE_Q203_7(Q203.7)";
  ELSE
      OLine8 := " ";
  END_CASE	

    Out_Visibility_1:=TRUE;

   CASE OP_Arr_OP10B_JB[Output_Page_num] OF
	200:  Out_Lamp1:=O10B_HPR_MTR_FWD_Q200_0;
	201:  Out_Lamp1:=O10B_BDY_BOWL_ON_Q201_0;
	202:  Out_Lamp1:=O10B_SPARE_Q202_0;
	203:  Out_Lamp1:=O10B_SPARE_Q203_0;
   ELSE
       Out_Visibility_1:=FALSE;	
   END_CASE
   
    Out_Visibility_2:=TRUE;
   
   CASE OP_Arr_OP10B_JB[Output_Page_num] OF
	200:  Out_Lamp2:=O10B_HPR_RST_Q200_1;
	201:  Out_Lamp2:=O10B_BDY_LNR_FEED1_ON_Q201_1;
	202:  Out_Lamp2:=O10B_SPARE_Q202_1;
	203:  Out_Lamp2:=O10B_SPARE_Q203_1;
   ELSE
       Out_Visibility_2:=FALSE;	
   END_CASE 
   
    Out_Visibility_3:=TRUE;
	
   CASE OP_Arr_OP10B_JB[Output_Page_num] OF
	200:  Out_Lamp3:=O10B_EXT_SPEED_Q200_2; 
	201:  Out_Lamp3:=O10B_BDY_LNR_FEED2_ON_Q201_2; 
	202:  Out_Lamp3:=O10B_SPARE_Q202_2; 
	203:  Out_Lamp3:=O10B_SPARE_Q203_2; 
   ELSE
       Out_Visibility_3:=FALSE;
   END_CASE 
   
    Out_Visibility_4:=TRUE;
   
   CASE OP_Arr_OP10B_JB[Output_Page_num] OF
	200:  Out_Lamp4:=O10B_SPARE_Q200_3; 
	201:  Out_Lamp4:=O10B_BDY_LNR1_AIR_PURGE_Q201_3; 
	202:  Out_Lamp4:=O10B_SPARE_Q202_3; 
	203:  Out_Lamp4:=O10B_SPARE_Q203_3;  
   ELSE
       Out_Visibility_4:=FALSE;
   END_CASE 
   
    Out_Visibility_5:=TRUE;
	
    CASE OP_Arr_OP10B_JB[Output_Page_num] OF
	200:  Out_Lamp5:=O10B_HPR_DOOR_SELCTN_IND_Q200_4; 
	201:  Out_Lamp5:=O10B_BDY_LNR2_AIR_PURGE_Q201_4 ; 
	202:  Out_Lamp5:=O10B_SPARE_Q202_4; 
	203:  Out_Lamp5:=O10B_SPARE_Q203_4; 	 
   ELSE
       Out_Visibility_5:=FALSE;
   END_CASE 
   
    Out_Visibility_6:=TRUE;
	
   CASE OP_Arr_OP10B_JB[Output_Page_num] OF
	200:  Out_Lamp6:=O10B_HPR_TWR_LMP_RED_Q200_5; 
	201:  Out_Lamp6:=O10B_HPR_DOOR_OPN_Q201_5; 
	202:  Out_Lamp6:=O10B_SPARE_Q202_5; 
	203:  Out_Lamp6:=O10B_SPARE_Q203_5; 
   ELSE           
       Out_Visibility_6:=FALSE;
   END_CASE 
    
	Out_Visibility_7:=TRUE;
	
   CASE OP_Arr_OP10B_JB[Output_Page_num] OF
	200:  Out_Lamp7:=O10B_HPR_TWR_LMP_GREEN_Q200_6; 
	201:  Out_Lamp7:=O10B_SPARE_Q201_6; 
	202:  Out_Lamp7:=O10B_SPARE_Q202_6; 
	203:  Out_Lamp7:=O10B_SPARE_Q203_6;  
   ELSE 
       Out_Visibility_7:=FALSE;
   END_CASE 
   
    Out_Visibility_8:=TRUE;
   
   CASE OP_Arr_OP10B_JB[Output_Page_num] OF
	200:  Out_Lamp8:=O10B_SPARE_Q200_7;  
	201:  Out_Lamp8:=O10B_SPARE_Q201_7;  
	202:  Out_Lamp8:=O10B_SPARE_Q202_7;  
	203:  Out_Lamp8:=O10B_SPARE_Q203_7;   
   ELSE
       Out_Visibility_8:=FALSE;	
   END_CASE 
 6: CASE IP_Arr_OP90JB[Input_Page_num] OF
    500: Line1:=" I90_SPARE_I500_0(I500.0)       ";
    501: Line1:=" I90_CONV1_FWD(I501.0)          ";
    502: Line1:=" I90_CONV1_TRK3_CHO_MOD2(I502.0)";
    503: Line1:=" I90_CONV2_REV(I503.0)          ";
    504: Line1:=" I90_CONV2_TRK3_CHO_MOD1(I504.0)";
    505: Line1:=" I90_SPARE_I505_0(I505.0)       ";
    else
     Line1:=" ";
    end_case 
    
    CASE IP_Arr_OP90JB[Input_Page_num] OF
    500: Line2:="I90_HPR1_LOW_LVL_FB(I500.1)        ";
    501: Line2:="I90_VBF1_CONV1_TRK1_OVERFLW(I501.1)";
    502: Line2:="I90_SPARE_I502_1(I502.1)           ";
    503: Line2:="I90_CONV2_FWD(I503.1)              ";
    504: Line2:="I90_CONV2_TRK3_CHO_MOD2(I504.1)    ";
    505: Line2:="I90_SPARE_I505_1(I505.1)           ";
    else
     Line2:=" ";
    end_case 
    
    CASE IP_Arr_OP90JB[Input_Page_num] OF
    500: Line3:="I90_HPR1_SOL_DOOR_SW_FB(I500.2)    ";
    501: Line3:="I90_VBF1_CONV1_TRK2_OVERFLW(I501.2)";
    502: Line3:="I90_HPR2_LOW_LVL_FB(I502.2)        ";
    503: Line3:="I90_VBF1_CONV2_TRK1_OVERFLW(I503.2)";
    504: Line3:="I90_VBF1_CONV_TRK_OVERFLW_2(I504.2)";
    505: Line3:="I90_SPARE_I505_2(I505.2)           ";
    else
     Line3:=" ";
    end_case 
    
    CASE IP_Arr_OP90JB[Input_Page_num] OF
    500: Line4:="I90_BOWL1_RDY(I500.3)              ";
    501: Line4:="I90_CONV1_TRK1_CHO_MOD1(I501.3)    ";
    502: Line4:="I90_HPR2_SOL_DOOR_SW_FB(I502.3)    ";
    503: Line4:="I90_VBF1_CONV2_TRK2_OVERFLW(I503.3)";
    504: Line4:="I90_VBF2_CONV_TRK_OVERFLW_2(I504.3)";
    505: Line4:="I90_SPARE_I505_3(I505.3)           ";
    else
     Line4:=" ";
    end_case 
    
    CASE IP_Arr_OP90JB[Input_Page_num] OF
    500: Line5:="I90_BOWL1_LOW_LVL(I500.4)      ";
    501: Line5:="I90_CONV1_TRK1_CHO_MOD2(I501.4)";
    502: Line5:="I90_BOWL2_RDY(I502.4)          ";
    503: Line5:="I90_CONV2_TRK1_CHO_MOD1(I503.4)";
    504: Line5:="I90_SPARE_I504_4(I504.4)       ";
    505: Line5:="I90_SPARE_I505_4(I505.4)       ";
    else
     Line5:=" ";
    end_case 
    
    CASE IP_Arr_OP90JB[Input_Page_num] OF
    500: Line6:="I90_BOWL1_OFF_ON(I500.5)        ";
    501: Line6:="I90_CONV1_TRK2_CHO_MOD1(I501.5) ";
    502: Line6:="I90_BOWL2_LOW_LVL(I502.5)       ";
    503: Line6:="I90_CONV2_TRK1_CHO_MOD2(I503.5) ";
    504: Line6:="I90_SPARE_I504_5(I504.5)        ";
    505: Line6:="I90_SPARE_I505_5(I505.5)        ";
    else
     Line6:=" ";
    end_case 
    
    CASE IP_Arr_OP90JB[Input_Page_num] OF
    500: Line7:="I90_HPR1_OFF_ON(I500.6)        ";
    501: Line7:="I90_CONV1_TRK2_CHO_MOD2(I501.6)";
    502: Line7:="I90_BOWL2_OFF_ON(I502.6)       ";
    503: Line7:="I90_CONV2_TRK2_CHO_MOD1(I503.6)";
    504: Line7:="I90_SPARE_I504_6(I504.6)       ";
    505: Line7:="I90_SPARE_I505_6(I505.6)       ";
    else
     Line7:=" ";
    end_case 
    
    CASE IP_Arr_OP90JB[Input_Page_num] OF
    500: Line8:="I90_CONV1_REV(I500.7)           ";
    501: Line8:="I90_CONV1_TRK3_CHO_MOD1(I501.7) ";
    502: Line8:="I90_HPR2_OFF_ON(I502.7)         ";
    503: Line8:="I90_CONV2_TRK2_CHO_MOD2(I503.7) ";
    504: Line8:="I90_SPARE_I504_7(I504.7)        ";
    505: Line8:="I90_SPARE_I505_7(I505.7)        ";
    else
     Line8:=" ";
    END_CASE 
	
  Visibility_1:=TRUE;
   
   CASE IP_Arr_OP90JB[Input_Page_num] OF
	500: Lamp1:=I90_SPARE_I500_0 ;
	501: Lamp1:=I90_CONV1_FWDI501_0 ;
	502: Lamp1:=I90_CONV1_TRK3_CHO_MOD2I502_0 ;
	503: Lamp1:=I90_CONV2_REVI503_0;
	504: Lamp1:=I90_CONV2_TRK3_CHO_MOD1I504_0 ;
	505: Lamp1:=I90_SPARE_I505_0 ;
   ELSE
       Visibility_1:=FALSE;	
   END_CASE
   
   
   Visibility_2:=TRUE;
   
   CASE IP_Arr_OP90JB[Input_Page_num] OF
	500: Lamp2:=I90_HPR1_LOW_LVL_FBI500_1 ;
	501: Lamp2:=I90_VBF1_CONV1_TRK1_OVERFLWI501_1 ;
	502: Lamp2:=I90_SPARE_I502_1 ;
	503: Lamp2:=I90_CONV2_FWDI503_1;
	504: Lamp2:=I90_CONV2_TRK3_CHO_MOD2I504_1 ;
	505: Lamp2:=I90_SPARE_I505_1 ;
   ELSE
       Visibility_2:=FALSE;	
   END_CASE
   
   
    Visibility_3:=TRUE;
   
   CASE IP_Arr_OP90JB[Input_Page_num] OF
	500: Lamp3:=I90_HPR1_SOL_DOOR_SW_FBI500_2 ;
	501: Lamp3:=I90_VBF1_CONV1_TRK2_OVERFLWI501_2 ;
	502: Lamp3:=I90_HPR2_LOW_LVL_FBI502_2 ;
	503: Lamp3:=I90_VBF1_CONV2_TRK1_OVERFLWI503_2;
	504: Lamp3:=I90_VBF1_CONV_TRK_OVERFLW_2I504_2 ;
	505: Lamp3:=I90_SPARE_I505_2 ;
   ELSE
       Visibility_3:=FALSE;	
   END_CASE
   
   
    Visibility_4:=TRUE;
   
